// TwinCAT 3 PLC project Struckig
// Title: Struckig
// Company: Stefan Besler
// Author: Stefan Besler and contributers
// ProjectVersion: 0.6.0.0
// ProgramVersion: 3.1.4024.12
// CompilerDefines: ZEUGWERK_TWINCAT_3_1_4024_22
// project tree:
//   / Constants.TcGVL, ParameterList.TcGVL
//   Struckig/Block/ BlockInterval.TcDUT, Block.TcDUT
//   Struckig/BrakeProfile/ BrakeProfile.TcPOU
//   Struckig/ Integrate.TcPOU (not stored), Otg.TcPOU
//   Struckig/Math/ BubbleSortLreal.TcPOU, Ceil.TcPOU, LrealBits.TcPOU, LrealFromBits.TcPOU, Power.TcPOU, Power2.TcPOU, Cbrt.TcPOU, Roots.TcPOU
//   Struckig/Position/ PositionStep1.TcPOU, PositionStep2.TcPOU
//   Struckig/Profile/ ProfileDesc.TcPOU
//   Struckig/Profile/_DataTypes/ PositionExtremaDesc.TcDUT, ProfileDirection.TcDUT, ProfileJerkSigns.TcDUT, ProfileLimits.TcDUT
//   Struckig/Velocity/ VelocityStep1.TcPOU, VelocityStep2.TcPOU
//   Struckig/_DataTypes/ ControlInterfaceType.TcDUT, DiscretizationType.TcDUT, SynchronizationType.TcDUT, TrajectoryErrorCode.TcDUT, TrajectoryState.TcDUT

// ---- Struckig/Block/BlockInterval.TcDUT
/// Which times are possible for synchronization?
TYPE INTERNAL BlockInterval :
STRUCT
  IsUsed : BOOL;
  Left, Right : LREAL;
  Profile : ProfileDesc;
END_STRUCT
END_TYPE

// ---- Struckig/Block/Block.TcDUT
TYPE Block :
STRUCT
  p_min : ProfileDesc; // Save min Profile so that it doesn't need to be recalculated in Step2
  Tmin : LREAL; // [s]
  a, b : BlockInterval; // Max. 2 intervals can be blocked: called a and b with corresponding profiles, order does not matter  
END_STRUCT
END_TYPE

// ---- Struckig/Profile/_DataTypes/PositionExtremaDesc.TcDUT
TYPE PositionExtremaDesc :
STRUCT
  Minimum, Maximum : LREAL; // The extreme position
  Tmin, Tmax : LREAL;  // Time when the positions are reached
END_STRUCT
END_TYPE

// ---- Struckig/Profile/_DataTypes/ProfileDirection.TcDUT
{attribute 'qualified_only'}
{attribute 'strict'}
TYPE INTERNAL ProfileDirection :
(
  Up,
  Down
);
END_TYPE

// ---- Struckig/Profile/_DataTypes/ProfileJerkSigns.TcDUT
{attribute 'qualified_only'}
{attribute 'strict'}
TYPE ProfileJerkSigns :
(
	Uddu,
  Udud 
);
END_TYPE

// ---- Struckig/Profile/_DataTypes/ProfileLimits.TcDUT
{attribute 'qualified_only'}
{attribute 'strict'}
TYPE ProfileLimits :
(
	Acc0Acc1Vel,
  Vel, 
  Acc0,
  Acc1,
  Acc0Acc1,
  Acc0Vel,
  Acc1Vel,
  None
);
END_TYPE

// ---- Struckig/_DataTypes/ControlInterfaceType.TcDUT
{attribute 'qualified_only'}
{attribute 'strict'}
TYPE ControlInterfaceType :
(
  Position, // Position-control: Full control over the entire kinematic state (Default)
  Velocity // Velocity-control: Ignores the current position, target position, and velocity limits
);
END_TYPE

// ---- Struckig/_DataTypes/DiscretizationType.TcDUT
{attribute 'qualified_only'}
{attribute 'strict'}
TYPE DiscretizationType :
(
  Continuous, /// Every trajectory synchronization duration is allowed (Default)
  Discrete /// The trajectory synchronization duration must be a multiple of the control cycle
);
END_TYPE

// ---- Struckig/_DataTypes/SynchronizationType.TcDUT
{attribute 'qualified_only'}
{attribute 'strict'}
TYPE SynchronizationType :
(
  Undefined,
  Phase, // Phase synchronize the DoFs when possible, else fallback to "Time" strategy
  TimeSync, // Always synchronize the DoFs to reach the target at the same time (Default)
  TimeIfNecessarySync, // Synchronize only when necessary (e.g. for non-zero target velocity or acceleration)
  None // Calculate every DoF independently
);
END_TYPE

// ---- Struckig/_DataTypes/TrajectoryErrorCode.TcDUT
{attribute 'qualified_only'}
TYPE TrajectoryErrorCode :
(
	Undefined := 0,
  InvalidInput,
  SynchronizationFailed,
  CalculateStep1Failed
);
END_TYPE

// ---- Struckig/_DataTypes/TrajectoryState.TcDUT
{attribute 'qualified_only'}
{attribute 'strict'}
TYPE TrajectoryState :
(
  Undefined,
  Idle,
  Busy,
  Error
);
END_TYPE

// ---- Constants.TcGVL
{attribute 'qualified_only'}
VAR_GLOBAL INTERNAL CONSTANT
  BrakeEpsilon : LREAL := 2.2E-14;
  DoubleEpsilon : LREAL := 2.2204460492503131E-016; // smallest such that 1.0+Constants.DoubleEpsilon != 1.0
  DoubleEpsilonSqrt : LREAL := 1.483E-8;
  Epsilon : LREAL := 1E-8;
  Epsilon16 : LREAL := 16 * 1E-8;
  EpsilonColinear : LREAL := 1E-7;
  Infinity : LREAL := 1.7976931348623157E+308;  
  Tolerance : LREAL := 1E-14;
  Cos120 : LREAL := -0.50;
  Sin120 : LREAL := 0.866025403784438646764;  
  Pi : LREAL := 3.14159265358979323846;
  Minimum : LREAL := 1.17549435082E-38;  // used for validating input
END_VAR

// ---- ParameterList.TcGVL
{attribute 'qualified_only'}
VAR_GLOBAL CONSTANT
  MaxDoFs : INT := 7;
  MaxIterations : BYTE := 127; // Maximum iterations when [shrinking an interval](xref:Struckig.Roots#ShrinkInterval)
  NumericalRobust : BOOL := TRUE;
END_VAR

// ---- Struckig/Math/Roots.TcPOU
PROGRAM INTERNAL Roots
VAR
  a2, aover3, q, r2, q3, aa, t : LREAL;
  a, b, c, d, rr, theta, ux, uyi, inva, invaa, bb, bover3a, p, halfq, yy, inv2b, x, y, uuu, vvv, www, w, h : LREAL;
  discriminant : LREAL;
  e0, e1, q1, q2, p1, p2, dd, sqrtD  : LREAL;
  a3, b3, c3 : LREAL;
  x3 : ARRAY[0..2] OF LREAL;
  iZeroes : INT;  
  deriv : ARRAY[0 .. 10] OF LREAL;
  fl, fh, temp : LREAL;
  dxold, dx, f,df : LREAL;
  j : INT;
  xn : LREAL;
  iterations : BYTE;
END_VAR

METHOD PolyDeri
VAR_INPUT
  coeffs : POINTER TO LREAL;
  coeffsCount : BYTE;
  out : POINTER TO LREAL;
END_VAR
FOR j:=0 TO coeffsCount DO
  out[j] := (coeffsCount - j) * coeffs[j];
END_FOR
END_METHOD

METHOD PolyEval : LREAL;
VAR_INPUT
  polynom : POINTER TO LREAL;
  degree : INT;
  x : LREAL;
END_VAR
IF degree > 0 THEN
  IF (ABS(x) < Constants.DoubleEpsilon) THEN
      PolyEval := polynom[degree];
  ELSIF (x = 1.0) THEN
    FOR j:= degree TO 0 BY -1
    DO
      PolyEval := PolyEval + polynom[j];
    END_FOR
  ELSE
    xn := 1.0;
    FOR j:= degree TO 0 BY -1 
    DO
      PolyEval := PolyEval + polynom[j] * xn;
      xn := xn * x;
    END_FOR
  END_IF
END_IF
END_METHOD

METHOD PolyMonicDeri
VAR_INPUT
  monic_coeffs : POINTER TO LREAL;
  coeffsCount : BYTE;
  out : POINTER TO LREAL;  
END_VAR
VAR
  i : BYTE;
END_VAR
out[0] := 1.0;
FOR i:=1 TO coeffsCount-1 DO
  out[i] := (coeffsCount- i) * (monic_coeffs[i] / (coeffsCount));
END_FOR
END_METHOD

// Calculate a single zero of polynom p(x) inside [lbound, ubound]
// Requirements: p(lbound)*p(ubound) < 0, lbound < ubound
METHOD ShrinkInterval : LREAL
VAR_INPUT
  p : POINTER TO LREAL;
  degree : BYTE;  
  l, h : LREAL;
END_VAR
PolyDeri(p, degree, out:=ADR(deriv));
fl := PolyEval(p, degree, l);
fh := PolyEval(p, degree, h);
IF (fl = 0.0) THEN
  ShrinkInterval := l;
  RETURN;
END_IF

IF (fh = 0.0) THEN
  ShrinkInterval := h;
  RETURN;
END_IF

IF (fl > 0.0)
THEN
  // swap l and h
  temp := l;
  l := h;
  h := temp;
END_IF

ShrinkInterval := (l + h) / 2;
dxold := ABS(h - l);
dx := dxold;
f := PolyEval(p, degree, ShrinkInterval);
df := PolyEval(ADR(deriv), degree-1, ShrinkInterval);
FOR iterations:=0 TO ParameterList.MaxIterations DO
  IF ((((ShrinkInterval - h) * df - f) * ((ShrinkInterval - l) * df - f) > 0.0) OR_ELSE (ABS(2 * f) > ABS(dxold * df))) THEN
    dxold := dx;
    dx := (h - l) / 2;
    ShrinkInterval := l + dx;
    IF (l = ShrinkInterval) THEN
      RETURN;
    END_IF
  ELSE
    dxold := dx;
    dx := f / df;
    temp := ShrinkInterval;
    ShrinkInterval := ShrinkInterval - dx;
    IF (temp = ShrinkInterval) THEN
      RETURN;
    END_IF
  END_IF
  
  IF (ABS(dx) < Constants.Tolerance) THEN
    RETURN;
  END_IF
  
  f := PolyEval(p, degree, ShrinkInterval);
  df := PolyEval(ADR(deriv), degree-1, ShrinkInterval);
  IF (f < 0.0) THEN
    l := ShrinkInterval;
  ELSE
    h := ShrinkInterval;
  END_IF
END_FOR
END_METHOD

METHOD SolveCub
VAR_INPUT
  polynom : POINTER TO LREAL;
END_VAR
VAR_IN_OUT
  rootCount : INT;
  roots : ARRAY[0..6] OF LREAL;
END_VAR
rootCount := -1;
a := polynom[0];
b := polynom[1];
c := polynom[2];
d := polynom[3];

IF (ABS(d) < Constants.DoubleEpsilon)
THEN
  // First solution is x = 0
  roots[0] := 0.0;
  rootCount := 1;
  
  // Converting to a quadratic equation
  d := c;
  c := b;
  b := a;
  a := 0.0;
END_IF

IF (ABS(a) < Constants.DoubleEpsilon)
THEN
  IF (ABS(b) < Constants.DoubleEpsilon)
  THEN
    // Linear equation
    h := (-d / c);
    IF ABS(c) > Constants.DoubleEpsilon AND_THEN h >= 0
    THEN
      roots[rootCount+1] := h;
      rootCount := rootCount + 1;
    END_IF
  ELSE
    // Quadratic equation
    discriminant := c * c - 4 * b * d;
    IF (discriminant >= 0)
    THEN
      inv2b := 1.0 / (2 * b);
      y := SQRT(discriminant);
      
      h := ((-c + y) * inv2b);
      IF h >= 0
      THEN
        roots[rootCount+1] := h;
        rootCount := rootCount + 1;
			END_IF
      
      h := ((-c - y) * inv2b);
      IF h >= 0
      THEN      
        roots[rootCount+1] := ((-c - y) * inv2b);
        rootCount := rootCount + 1;
      END_IF
      
    END_IF
  END_IF

ELSE
  
  // Cubic equation
  inva := 1.0 / a;
  invaa := inva * inva;
  bb := b * b;
  bover3a := b * inva / 3;
  p := (a * c - bb / 3) * invaa;
  halfq := (2 * bb * b - 9 * a * b * c + 27 * a * a * d) * (0.5 / 27) * invaa * inva;
  yy := p * p * p / 27 + halfq * halfq;  
    
  IF (yy > Constants.DoubleEpsilon) THEN
    // Sqrt is positive: one real solution}
    y := SQRT(yy);
    uuu := -halfq + y;
    vvv := -halfq - y;
    www := SEL(ABS(uuu) > ABS(vvv), vvv, uuu);
    w := cbrt(www);
    
    h := (w - p / (3 * w) - bover3a);
    IF h >= 0
    THEN
      roots[rootCount+1] := h;
      rootCount := rootCount + 1;    
		END_IF

  ELSIF (yy < -Constants.DoubleEpsilon) THEN
    // Sqrt is negative: three real solutions
    x := -halfq;
    y := SQRT(-yy);

    // Convert to polar form}
    IF ABS(x) > Constants.DoubleEpsilon THEN
      theta := SEL((x > 0.0), (ATAN(y / x) + Constants.Pi), ATAN(y / x));
      rr := SQRT(x * x - yy);
    ELSE
      // Vertical line}
      theta := Constants.Pi / 2;
      rr := y;
    END_IF
    
    // Calculate cube root
    theta := theta / 3;
    rr := 2 * cbrt(rr);
    // Convert to complex coordinate
    ux := COS(theta) * rr;
    uyi := SIN(theta) * rr;
    // First solution
    h := (ux - bover3a);
    IF h >= 0
    THEN
      roots[rootCount+1] := h;
      rootCount := rootCount + 1;
		END_IF
    
    // Second solution, rotate +120 degrees
    h := ux * Constants.Cos120 - uyi * Constants.Sin120 - bover3a;
    IF h >= 0
    THEN
      roots[rootCount+1] := h;
      rootCount := rootCount + 1;
		END_IF
    
    // Third solution, rotate -120 degrees
    h := ux * Constants.Cos120 + uyi * Constants.Sin120 - bover3a;
    IF h >= 0
    THEN
      roots[rootCount+1] := h;
      rootCount := rootCount + 1;
		END_IF
  ELSE
    // Sqrt is zero: two real solutions
    www := -halfq;
    w := 2 * cbrt(www);
    // First solution
    h := (w - bover3a);
    IF h >= 0
    THEN
      roots[rootCount+1] := h;
      rootCount := rootCount + 1;
		END_IF
    
    // Second solution, rotate +120 degrees
    h := (w * Constants.Cos120 - bover3a);
    IF h >= 0
    THEN
      roots[rootCount+1] := h;
      rootCount := rootCount + 1;
		END_IF
  END_IF
END_IF
END_METHOD

/// Calculate all roots of the monic quartic equation: x^4 + a*x^3 + b*x^2 + c*x + d = 0
METHOD SolveQuartMonic
VAR_INPUT
  polynom : POINTER TO LREAL;  
  degree : LREAL;
END_VAR
VAR_IN_OUT
  rootCount : INT;
  roots : ARRAY[0..6] OF LREAL;
END_VAR
rootCount := -1;

a := polynom[0];
b := polynom[1];
c := polynom[2];
d := polynom[3];
e0 := cbrt(c * c);
IF (ABS(a) < Constants.DoubleEpsilon AND_THEN ABS(b) < Constants.DoubleEpsilonSqrt AND_THEN ABS(c) < Constants.DoubleEpsilonSqrt AND_THEN ABS(d) < Constants.DoubleEpsilon) AND_THEN
   ABS(e0) > Constants.DoubleEpsilon
THEN
  e1 := (b * b + 12 * d)/(9 * e0);
  q1 := -(4 * b) / 3 - e0 - e1;
  p1 := SQRT(-q1 - 2 * b);
  q2 := 2 * c / p1;
  
  dd := q1 - q2;
  IF (dd > 0.0)
  THEN  
    sqrtD := SQRT(dd);
    
    h := ((p1 + sqrtD) / 2);
    IF h >= 0
    THEN
      roots[0] := h;
      rootCount := 0;
		END_IF
    
    h := ((p1 - sqrtD) / 2);
    IF h >= 0
    THEN
      roots[rootCount+1] := h;
      rootCount := rootCount + 1;
		END_IF
  END_IF
  
  dd := q1 + q2;
  IF (dd > 0.0)
  THEN  
    sqrtD := SQRT(dd);
    
    h := ((-p1 + sqrtD) / 2);
    IF h >= 0
    THEN
      roots[rootCount+1] := h;
      rootCount := rootCount + 1;
		END_IF
    
    h := ((-p1 - sqrtD) / 2);
    IF h >= 0
    THEN
      roots[rootCount+1] := h;
      rootCount := rootCount + 1;
		END_IF
  END_IF
  RETURN;
END_IF

IF (ABS(c) < Constants.DoubleEpsilon AND_THEN ABS(d) < Constants.DoubleEpsilon)
THEN
  roots[0] := 0.0;
  rootCount := rootCount+1;
  
  dd := a * a - 4 * b;
  IF (ABS(dd) < Constants.DoubleEpsilon)
  THEN
    h := (-a / 2);
    IF h >= 0
    THEN
      roots[rootCount+1] := h;
      rootCount := rootCount + 1;
		END_IF
  ELSIF (dd > 0)
  THEN
    sqrtD := SQRT(dd);
    h := ((-a - sqrtD) / 2);
    IF h >= 0
    THEN
      roots[rootCount+1] := h;
      rootCount := rootCount + 1;
		END_IF
    
    h := ((-a + sqrtD) / 2);
    IF h >= 0
    THEN
      roots[rootCount+1] := h;
      rootCount := rootCount + 1;
		END_IF  
  END_IF
  RETURN;
END_IF

a3 := -b;
b3 := a * c - 4 * d;
c3 := -a * a * d - c * c + 4 * b * d;

// Solve the resolvent: y^3 - b*y^2 + (ac - 4*d)*y - a^2*d - c^2 + 4*b*d = 0
iZeroes := SolveResolvent(ADR(x3), a3, b3, c3);

y := x3[0];
// Choosing Y with maximal absolute value.
IF (iZeroes <> 1) THEN
  IF ABS(x3[1]) > ABS(y) THEN
    y := x3[1];
  END_IF
  
  IF ABS(x3[2]) > ABS(y) THEN
    y := x3[2];
  END_IF
END_IF

// h1 + h2 = y AND_THEN h1*h2 = d  <=>  h^2 - y*h + d = 0    (h === q)
dd := y * y - 4 * d;
IF (ABS(dd) < Constants.DoubleEpsilon) THEN
  q1 := q2 := y / 2;
  // g1 + g2 = a AND_THEN g1 + g2 = b - y   <=>   g^2 - a*g + b - y = 0    (p === g)}
  dd := a * a - 4 * (b - y);
  IF (ABS(dd) < Constants.DoubleEpsilon) THEN
    p1 := p2 := a / 2;
  ELSE
    sqrtD := SQRT(dd);
    p1 := (a + sqrtD) / 2;
    p2 := (a - sqrtD) / 2;
  END_IF
ELSE
  sqrtD := SQRT(dd);
  q1 := (y + sqrtD) / 2;
  q2 := (y - sqrtD) / 2;
  // g1 + g2 = a AND_THEN g1*h2 + g2*h1 = c   ( AND_THEN g === p )  Krammer
  p1 := (a * q1 - c) / (q1 - q2);
  p2 := (c - a * q2) / (q1 - q2);
END_IF

// Solve the quadratic equation: x^2 + p1*x + q1 = 0
dd := p1 * p1 - 4 * q1;
IF (ABS(dd) < Constants.Epsilon16) THEN
  
  h:= (-p1 / 2);
  IF h >= 0
  THEN
    roots[rootCount+1] := h;
    rootCount := rootCount + 1;
  END_IF
  
ELSIF (dd > 0.0)  THEN
  sqrtD := SQRT(dd);
  h := ((-p1 + sqrtD) / 2);
  IF h >= 0
  THEN
    roots[rootCount+1] := h;
    rootCount := rootCount + 1;
  END_IF
    
  h := ((-p1 - sqrtD) / 2);
  IF h >= 0
  THEN
    roots[rootCount+1] := h;
    rootCount := rootCount + 1;
  END_IF
END_IF

// Solve the quadratic equation: x^2 + p2*x + q2 = 0
dd := p2 * p2 - 4 * q2;
IF (ABS(dd) < Constants.Epsilon16) THEN
  h := (-p2 * 0.5);
  IF h >= 0
  THEN
    roots[rootCount+1] := h;
    rootCount := rootCount + 1;
  END_IF  
ELSIF (dd > 0.0) THEN
  sqrtD := SQRT(dd);
  h := ((-p2 + sqrtD) / 2); 
  IF h >= 0
  THEN
    roots[rootCount+1] := h;
    rootCount := rootCount + 1;
  END_IF
  
  h := ((-p2 - sqrtD) / 2);
  IF h >= 0
  THEN
    roots[rootCount+1] := h;
    rootCount := rootCount + 1;
  END_IF
END_IF
END_METHOD

/// Solve resolvent eqaution of corresponding Quartic equation
/// The input x must be of length 3
/// Number of zeros are returned
METHOD SolveResolvent : INT
VAR_INPUT
  x : POINTER TO LREAL;
  a,b,c : LREAL;
END_VAR
aover3 := a / 3;
a2 := a * a;
q := (a2 - 3 * b) / 9;
rr := a * (2 * a2 - 9 * b) / 54 + c / 2;
r2 := rr * rr;
q3 := q * q * q;

IF (r2 < q3) THEN
  t := rr / SQRT(q3);
  IF (t < -1.0) THEN
      t := -1.0;
  END_IF
  
  IF (t > 1.0) THEN
      t := 1.0;
  END_IF
  
  q := -2 * SQRT(q);
  theta := ACOS(t) / 3;
  ux := COS(theta) * q;
  uyi := SIN(theta) * q;
  x[0] := ux - aover3;
  x[1] := ux * Constants.Cos120 - uyi * Constants.Sin120 - aover3;
  x[2] := ux * Constants.Cos120 + uyi * Constants.Sin120 - aover3;
  SolveResolvent := 3;
  RETURN;

ELSE
  aa := -cbrt(ABS(rr) + SQRT(r2 - q3));
  IF (rr < 0.0) THEN
    aa := -aa;
  END_IF
  bb := SEL(0.0 = aa, q / aa, 0.0);
  
  x[0] := (aa + bb) - aover3;
  x[1] := -(aa + bb) / 2 - aover3;
  x[2] := SQRT(3) * (aa - bb) / 2;
  IF (ABS(x[2]) < Constants.DoubleEpsilon) THEN
    x[2] := x[1];
    SolveResolvent := 2;
    RETURN;
  END_IF
  
  SolveResolvent := 1;
END_IF
END_METHOD

END_PROGRAM

// ---- Struckig/Math/Cbrt.TcPOU
/// The TwinCAT code is a modified version of the original C code from
/// http://www.netlib.org/fdlibm/s_cbrt.c and came with this notice.
///
/// ```
/// Copyright (C) 1993 by Sun Microsystems, Inc. All rights reserved.
///
/// Developed at SunSoft, a Sun Microsystems, Inc. business.
/// Permission to use, copy, modify, and distribute this
/// software is freely granted, provided that this notice
/// is preserved.
/// ```
///
///
/// Small modifications were made, while the original code said
/// ```
/// chop to 20 bits, make larger than cbrt(x)
/// t := LrealFromBits((LrealBits(t) AND SHL(H, 28)) + SHL(J, 30));
/// ```
/// Modern compilers seem to round t away from 0 to 23 bits.
/// see https://github.com/stdlib-js/math-base-special-cbrt/blob/main/src/cbrt.c
FUNCTION Cbrt : LREAL
VAR_INPUT
  x : LREAL;
END_VAR
VAR CONSTANT
  B1 : ULINT := 715094163;                  // (682-0.03306235651)*2**20
  B2 : ULINT := 696219795;                  // (664-0.03306235651)*2**20
  C : LREAL := 5.42857142857142815906E-01;  // 19/35     = 0x3FE15F15F15F15F1
  D : LREAL := -7.05306122448979611050E-01; // -864/1225 = 0xBFE691DE2532C834
  E : LREAL := 1.41428571428571436819E+00;  // 99/70     = 0x3FF6A0EA0EA0EA0F
  F : LREAL := 1.60714285714285720630E+00;  // 45/28     = 0x3FF9B6DB6DB6DB6E
  G : LREAL := 3.57142857142857150787E-01;  // 5/14      = 0x3FD6DB6DB6DB6DB7
  J : ULINT := 1;
  Mask : ULINT := ULINT#16#FFFFFFFFC0000000;
  AMask : ULINT := ULINT#16#80000000;
  SmallestNormal : LREAL := 2.22507385850720138309E-308; // 2**-1022  = 0x0010000000000000  
END_VAR
VAR
  sign : BOOL;
  t, r1, s1, w : LREAL;
END_VAR

// test x=0 and x=NaN
IF x = 0 OR_ELSE x <> x
THEN
  Cbrt := x;
  RETURN;
END_IF

sign := FALSE;
IF x < 0
THEN
  x := -x;
  sign := TRUE;  
END_IF

// rough cbrt to 5 bits
t := LrealFromBits(LrealBits(x)/3 + SHL(B1, 32));
IF x < SmallestNormal
THEN
  // subnormal number
  t := LrealFromBits(SHL(J, 54)); // set t= 2**54
  t := t * x;
  t := LrealFromBits(LrealBits(t)/3 + SHL(B2, 32));
END_IF

// new cbrt to 23 bits
r1 := t * t / x;
s1 := C + r1*t;
t := t * (G + F/(s1+E+D/s1));

// see https://github.com/stdlib-js/math-base-special-cbrt/blob/main/src/cbrt.c
t := LrealFromBits((LrealBits(t) + AMask) AND Mask);

// one step newton iteration to 53 bits with error less than 0.667ulps
s1 := t * t; // t*t is exact
r1 := x / s1;
w := t + t;
r1 := (r1 - t) / (w + r1); // r-s is exact
t := t + t*r1;

// restore the sign bit
IF sign
THEN
  t := -t;
END_IF

Cbrt := t;
    
// this one is a bit more prone to numerical errors
// Cbrt := SEL(x < 0, 1.0, -1.0) * EXPT(ABS(x), 1.0 / 3.0);

END_FUNCTION

// ---- Struckig/Math/LrealFromBits.TcPOU
{attribute 'hide'}
FUNCTION LrealFromBits : LREAL
VAR_INPUT
  b : ULINT;
END_VAR
VAR
  x : POINTER TO LREAL := ADR(b);
END_VAR

LrealFromBits := x^;

END_FUNCTION

// ---- Struckig/Math/LrealBits.TcPOU
{attribute 'hide'}
FUNCTION LrealBits : ULINT
VAR_INPUT
  x : LREAL;
END_VAR
VAR
  b : POINTER TO ULINT := ADR(x);
END_VAR

LrealBits := b^;

END_FUNCTION

// ---- Struckig/BrakeProfile/BrakeProfile.TcPOU
/// Calculates (pre- or post-) profile to get current or final state below the limits
FUNCTION_BLOCK BrakeProfile
VAR_INPUT
  Duration : LREAL; //! Overall duration
  t, j, a, v, p : ARRAY[0..1] OF LREAL; //! Profile information for a two-step profile  
  IsUsed : BOOL;
END_VAR
VAR
  t_to_a_min, t_to_a_max, t_min_to_v_max, t_to_a_zero, t_to_v_min, t_to_v_max : LREAL;
  t_to_v_max_with_constant, t_to_v_min_with_constant, v_at_a0, v_at_a_max, v_at_a_min : LREAL;
END_VAR

METHOD AccelerationBrake
VAR_INPUT
  v0, a0 : LREAL;
  vMax, vMin : LREAL;
  aMax, aMin : LREAL;
  jMax : LREAL;
END_VAR
VAR_IN_OUT
  t_brake : ARRAY[0..1] OF LREAL;
  j_brake : ARRAY[0..1] OF LREAL;    
END_VAR
j_brake[0] := -jMax;

t_to_a_max := (a0 - aMax) / jMax;
t_to_a_zero := a0 / jMax;

v_at_a_max := VelocityAtTime(v0, a0, -jMax, t_to_a_max);
v_at_a0 := VelocityAtTime(v0, a0, -jMax, t_to_a_zero);

IF (v_at_a0 > vMax AND_THEN jMax > 0) OR_ELSE (v_at_a0 < vMax AND_THEN jMax < 0)
THEN
  VelocityBrake(v0, a0, vMax, vMin, aMax, aMin, jMax, t_brake, j_brake);

ELSIF (v_at_a_max < vMin AND_THEN jMax > 0) OR_ELSE (v_at_a_max > vMin AND_THEN jMax < 0)
THEN
  t_to_v_min := -(v_at_a_max - vMin)/aMax;
  t_to_v_max := -aMax/(2*jMax) - (v_at_a_max + vMax)/aMax;
  t_brake[0] := t_to_a_max + Constants.BrakeEpsilon;
  t_brake[1] := MAX(MIN(t_to_v_min, v_at_a_max - Constants.BrakeEpsilon), 0.0);
ELSE
  t_brake[0] := t_to_a_max + Constants.BrakeEpsilon;
END_IF
END_METHOD

METHOD PositionBrakeTrajectory
VAR_INPUT
  v0, a0 : LREAL;
  vMax, vMin : LREAL;
  aMax, aMin : LREAL;
  jMax : LREAL;
END_VAR
VAR_IN_OUT
  t_brake : ARRAY[0..1] OF LREAL;
  j_brake : ARRAY[0..1] OF LREAL;    
END_VAR
t_brake[0] := 0.0;
t_brake[1] := 0.0;
j_brake[0] := 0.0;
j_brake[1] := 0.0;

IF a0 > aMax
THEN
  AccelerationBrake(v0, a0, vMax, vMin, aMax, aMin, jMax, t_brake, j_brake);
ELSIF a0 < aMin
THEN
  AccelerationBrake(v0, a0, vMin, vMax, aMin, aMax, -jMax, t_brake, j_brake);
ELSIF ((v0 > vMax AND_THEN VelocityAtZeroAcceleration(v0, a0, -jMax) > vMin) OR_ELSE (a0 > 0 AND_THEN VelocityAtZeroAcceleration(v0, a0, jMax) > vMax))
THEN
  VelocityBrake(v0, a0, vMax, vMin, aMax, aMin, jMax, t_brake, j_brake);
ELSIF ((v0 < vMin AND_THEN VelocityAtZeroAcceleration(v0, a0, jMax) < vMax) OR_ELSE (a0 < 0 AND_THEN VelocityAtZeroAcceleration(v0, a0, -jMax) < vMin))
THEN
  VelocityBrake(v0, a0, vMin, vMax, aMin, aMax, -jMax, t_brake, j_brake);      
END_IF
END_METHOD

METHOD VelocityAtTime : LREAL
VAR_INPUT
  v0, a0 : LREAL;
  j : LREAL;
  t : LREAL;
END_VAR
VelocityAtTime := v0 + t * (a0 + j * t * 0.5);
END_METHOD

METHOD VelocityAtZeroAcceleration : LREAL
VAR_INPUT
  v0, a0 : LREAL;
  j : LREAL;
END_VAR
VelocityAtZeroAcceleration := v0 + (a0 * a0) / (2 * j);
END_METHOD

METHOD VelocityBrake
VAR_INPUT
  v0, a0 : LREAL;
  vMax, vMin : LREAL;
  aMax, aMin : LREAL;
  jMax : LREAL;
END_VAR
VAR_IN_OUT
  t_brake : ARRAY[0..1] OF LREAL;
  j_brake : ARRAY[0..1] OF LREAL;    
END_VAR
j_brake[0] := -jMax;
t_to_a_min := (a0 - aMin)/jMax;
t_to_v_max := a0*a0 + 2 * jMax * (v0 - vMax);
t_to_v_min := a0*a0 / 2 + jMax * (v0 - vMin);

IF t_to_v_max < 0 OR_ELSE t_to_v_min < 0
THEN
  RETURN;
END_IF

t_to_v_max := a0/jMax + SQRT(t_to_v_max) / ABS(jMax);
t_to_v_min := a0/jMax + SQRT(t_to_v_min) / ABS(jMax);
t_min_to_v_max := MIN(t_to_v_max, t_to_v_min);

IF (t_to_a_min < t_min_to_v_max)
THEN
  v_at_a_min := VelocityAtTime(v0, a0, -jMax, t_to_a_min);
  t_to_v_max_with_constant := -(v_at_a_min - vMax)/aMin;
  t_to_v_min_with_constant := -0.5*aMin/jMax - (v_at_a_min - vMin)/aMin;
  t_brake[0] := t_to_a_min - Constants.BrakeEpsilon;
  t_brake[1] := MAX(MIN(t_to_v_max_with_constant, t_to_v_min_with_constant), 0.0);
ELSE
  t_brake[0] := t_min_to_v_max - Constants.BrakeEpsilon;
END_IF
END_METHOD

METHOD VelocityBrakeTrajectory
VAR_INPUT
  v0, a0 : LREAL;
  aMax, aMin : LREAL;
  jMax : LREAL;
END_VAR
VAR_IN_OUT
  t_brake : ARRAY[0..1] OF LREAL;
  j_brake : ARRAY[0..1] OF LREAL;    
END_VAR
t_brake[0] := 0.0;
t_brake[1] := 0.0;
j_brake[0] := 0.0;
j_brake[1] := 0.0;

IF (a0 > aMax)
THEN
  j_brake[0] := -jMax;
  t_brake[0] := (a0 - aMax)/jMax + Constants.BrakeEpsilon;
ELSIF (a0 < aMin)
THEN
  j_brake[0] := jMax;
  t_brake[0] := -(a0 - aMin)/jMax + Constants.BrakeEpsilon;
END_IF
END_METHOD

END_FUNCTION_BLOCK

// ---- Struckig/Math/BubbleSortLreal.TcPOU
FUNCTION BubbleSortLreal : BOOL
VAR_INPUT
  data : POINTER TO LREAL; // input unsorted array
  size : INT; // elements in the data array
  indicesSorted : POINTER TO INT; // actual output, sorted indices
END_VAR
VAR
  i, j, h : INT;
END_VAR

FOR i:=0 TO size
DO
  indicesSorted[i] := i;
END_FOR

// Bubblesort possible_t_syncs from best to worst
FOR i:=0 TO size-1
DO
  FOR j:=0 TO size-1-i
  DO  
    IF data[indicesSorted[j]] > data[indicesSorted[j+1]]
    THEN
      h := indicesSorted[j];
      indicesSorted[j] := indicesSorted[j+1];
      indicesSorted[j+1] := h;     
		END_IF
  END_FOR
END_FOR

END_FUNCTION

// ---- Struckig/Math/Ceil.TcPOU
FUNCTION Ceil : LREAL
VAR_INPUT
  val : LREAL;
END_VAR
VAR CONSTANT
  InfinityBits : ULINT := ULINT#16#7FF0000000000000;
END_VAR
VAR
  InfinityPtr : POINTER TO LREAL := ADR(InfinityBits);
END_VAR

IF val <> val OR_ELSE val = InfinityPtr^ OR_ELSE val = -InfinityPtr^ // nan or inf
THEN
  RETURN;
END_IF

Ceil := DINT_TO_LREAL(LREAL_TO_DINT(val));
IF Ceil < val THEN
	Ceil := Ceil + 1;
END_IF;

END_FUNCTION

// ---- Struckig/Math/Power.TcPOU
FUNCTION INTERNAL Power : LREAL
VAR_INPUT
  v : LREAL;
  e : LREAL;
END_VAR

Power := SEL(v < 0, 1.0, -1.0) * EXPT(ABS(v), e);

END_FUNCTION

// ---- Struckig/Math/Power2.TcPOU
FUNCTION INTERNAL Power2 : LREAL
VAR_INPUT
  v : LREAL;
END_VAR

Power2 := v*v;

END_FUNCTION

// ---- Struckig/Position/PositionStep1.TcPOU
FUNCTION_BLOCK INTERNAL PositionStep1
VAR
  p0, v0, a0 : LREAL;
  pf, vf, af : LREAL;
  _vMax, _vMin, _aMax, _aMin, _jMax : LREAL;

  // Pre-calculated expressions
  pd : LREAL;
  v0_v0, vf_vf : LREAL;
  a0_a0, a0_p3, a0_p4 : LREAL;
  af_af, af_p3, af_p4 : LREAL;
  jMax_jMax : LREAL;
  
  // runtime  calculated expressions
  polynom : ARRAY[0..4] OF LREAL;
  orig : LREAL;
  deriv : LREAL;
  t : LREAL;
  i : INT;
  h0, h1, h2, h2_h2, h3 : LREAL;
  t_min, t_max : LREAL;
  t_acc1, t_acc0 : LREAL;
  validProfiles : ARRAY[0..5] OF ProfileDesc; // Max 5 valid profiles + 1 spare for numerical issues
  validProfileCounter : INT := -1;
  
  rootCount : INT;
  root : ARRAY[0..6] OF LREAL;
  left_duration, right_duration : LREAL;   
END_VAR

METHOD AddInterval
VAR_INPUT
  interval : REFERENCE TO BlockInterval;
  Left : REFERENCE TO ProfileDesc;
  Right : REFERENCE TO ProfileDesc;
END_VAR
left_duration := Left.t_sum[6] + Left.Brake.Duration;
right_duration := Right.t_sum[6] + Right.Brake.Duration;
IF (left_duration < right_duration)
THEN
  interval.Left := left_duration;
  interval.Right := right_duration;
  interval.Profile := Right;
  interval.IsUsed := TRUE;
ELSE
  interval.Left := right_duration;
  interval.Right := left_duration;
  interval.Profile := Left;
  interval.IsUsed := TRUE;  
END_IF
END_METHOD

METHOD AddProfile
VAR_IN_OUT CONSTANT
  Profile : ProfileDesc;
  jMax : LREAL;
END_VAR
validProfileCounter := validProfileCounter + 1;
validProfiles[validProfileCounter] := Profile;
validProfiles[validProfileCounter].Direction := SEL(jMax > 0, ProfileDirection.Down, ProfileDirection.Up);
END_METHOD

METHOD CalculateBlock : BOOL
VAR_INPUT
  block : REFERENCE TO Block;
END_VAR
VAR
  i, j : INT;
  Tmin : LREAL;
  idx_min : INT;
  idx_else_1, idx_else_2, idx_else_3, idx_else_4 : INT;
END_VAR
IF validProfileCounter = 0
THEN
  block.Pmin := validProfiles[0];
  block.Tmin := block.Pmin.t_sum[6] + block.Pmin.Brake.Duration;  
  CalculateBlock := TRUE;

ELSIF validProfileCounter = 1 
THEN

  IF ABS(validProfiles[0].t_sum[6] - validProfiles[1].t_sum[6]) < 8*Constants.Epsilon
  THEN
    block.Pmin := validProfiles[0];
    block.Tmin := block.Pmin.t_sum[6] + block.Pmin.Brake.Duration;  
    CalculateBlock := TRUE;
    RETURN;
	END_IF
  
  IF ParameterList.NumericalRobust
  THEN
    idx_min := SEL(validProfiles[0].t_sum[6] < validProfiles[1].t_sum[6], 1, 0);
    idx_else_1 := (idx_min + 1) MOD 2;

    block.Pmin := validProfiles[idx_min];
    block.Tmin := block.Pmin.t_sum[6] + block.Pmin.Brake.Duration;
    
    AddInterval(block.A, validProfiles[idx_min], validProfiles[idx_else_1]);
    CalculateBlock := TRUE;
    RETURN; 
	END_IF

// Only happens due to numerical issues
ELSIF (validProfileCounter = 3) 
THEN
  // Find "identical" profiles
  IF (ABS(validProfiles[0].t_sum[6] - validProfiles[1].t_sum[6]) < 32*Constants.Epsilon AND_THEN validProfiles[0].Direction <> validProfiles[1].Direction)
  THEN
    RemoveProfile(1);
  ELSIF (ABS(validProfiles[2].t_sum[6] - validProfiles[3].t_sum[6]) < 256*Constants.Epsilon  AND_THEN validProfiles[2].Direction <> validProfiles[3].Direction)
  THEN
    RemoveProfile(3);
  ELSIF (ABS(validProfiles[0].t_sum[6] - validProfiles[3].t_sum[6]) < 256*Constants.Epsilon AND_THEN validProfiles[0].Direction <> validProfiles[3].Direction)
  THEN
    RemoveProfile(3);
  ELSE
    RETURN;
  END_IF

ELSIF ((validProfileCounter+1) MOD 2 = 0)
THEN
  RETURN;
END_IF

// Find index of fastest Profile
Tmin := Constants.Infinity;
FOR i:=0 TO validProfileCounter
DO
  FOR j:=0 TO validProfileCounter
  DO
    IF validProfiles[i].t_sum[6] + validProfiles[i].brake.Duration < validProfiles[j].t_sum[6] + validProfiles[j].brake.Duration AND_THEN
       validProfiles[i].t_sum[6] + validProfiles[i].brake.Duration < Tmin
    THEN
      Tmin := validProfiles[i].t_sum[6] + validProfiles[i].brake.Duration;
      idx_min := i;
		END_IF
  END_FOR
END_FOR

block.A.IsUsed := FALSE;
block.B.IsUsed := FALSE;
block.Pmin := validProfiles[idx_min];
block.Tmin := block.Pmin.t_sum[6] + block.Pmin.Brake.Duration;  

IF (validProfileCounter = 2)
THEN
  idx_else_1 := (idx_min + 1) MOD 3;
  idx_else_2 := (idx_min + 2) MOD 3;
  
  AddInterval(block.A, validProfiles[idx_else_1], validProfiles[idx_else_2]);
  CalculateBlock := TRUE;
  RETURN;

 ELSIF (validProfileCounter = 4)
 THEN
  idx_else_1 := (idx_min + 1) MOD 5;
  idx_else_2 := (idx_min + 2) MOD 5;
  idx_else_3 := (idx_min + 3) MOD 5;
  idx_else_4 := (idx_min + 4) MOD 5;
  
  IF (validProfiles[idx_else_1].Direction = validProfiles[idx_else_2].Direction)
  THEN
    AddInterval(block.A, validProfiles[idx_else_1], validProfiles[idx_else_2]);
    AddInterval(block.B, validProfiles[idx_else_3], validProfiles[idx_else_4]);
  ELSE 
    AddInterval(block.A, validProfiles[idx_else_1], validProfiles[idx_else_4]);
    AddInterval(block.B, validProfiles[idx_else_2], validProfiles[idx_else_3]);
  END_IF
  
  CalculateBlock := TRUE;
END_IF
END_METHOD

METHOD Get : BOOL
VAR_INPUT
  Profilefile : REFERENCE TO ProfileDesc;
  block : REFERENCE TO Block; 
END_VAR
VAR_INST
  vMax, vMin, aMax, aMin, jMax : LREAL;  
END_VAR
Profilefile.SetBoundaryPosition(p0, v0, a0, pf, vf, af);
validProfileCounter := -1;

IF (ABS(vf) < Constants.DoubleEpsilon AND_THEN ABS(af) < Constants.DoubleEpsilon) THEN
  vMax := SEL(pd >= 0, _vMin, _vMax);
  vMin := SEL(pd >= 0, _vMax, _vMin);
  aMax := SEL(pd >= 0, _aMin, _aMax);
  aMin := SEL(pd >= 0, _aMax, _aMin);
  jMax :=SEL (pd >= 0,-_jMax, _jMax);

  IF ABS(v0) < Constants.DoubleEpsilon AND_THEN ABS(a0) < Constants.DoubleEpsilon AND_THEN ABS(pd) < Constants.DoubleEpsilon
  THEN
    time_none(Profilefile, vMax, vMin, aMax, aMin, jMax);
  ELSE
    // There is no blocked interval when vf==0 && af==0, so return after first found profile
    time_all_vel(Profilefile, vMax, vMin, aMax, aMin, jMax);
    IF (validProfileCounter > 0) THEN
      Get := CalculateBlock(block);
      RETURN;
    END_IF
    time_none(Profilefile, vMax, vMin, aMax, aMin, jMax);
    IF (validProfileCounter > 0) THEN
      Get := CalculateBlock(block);
      RETURN;
    END_IF
    time_acc0(Profilefile, vMax, vMin, aMax, aMin, jMax);
    IF (validProfileCounter > 0) THEN
      Get := CalculateBlock(block);
      RETURN;
    END_IF
    time_acc1(Profilefile, vMax, vMin, aMax, aMin, jMax);
    IF (validProfileCounter > 0) THEN
      Get := CalculateBlock(block);
      RETURN;
    END_IF
    time_acc0_acc1(Profilefile, vMax, vMin, aMax, aMin, jMax);
    IF (validProfileCounter > 0) THEN
      Get := CalculateBlock(block);
      RETURN;
    END_IF
    time_all_vel(Profilefile, vMax, vMin, aMax, aMin, jMax);
    IF (validProfileCounter > 0) THEN
      Get := CalculateBlock(block);
      RETURN;
    END_IF
    time_none(Profilefile, vMin, vMax, aMin, aMax, -jMax);
    IF (validProfileCounter > 0) THEN
      Get := CalculateBlock(block);
      RETURN;
    END_IF
    time_acc0(Profilefile, vMin, vMax, aMin, aMax, -jMax);
    IF (validProfileCounter > 0) THEN
      Get := CalculateBlock(block);
      RETURN;
    END_IF
    time_acc1(Profilefile, vMin, vMax, aMin, aMax, -jMax);
    IF (validProfileCounter > 0) THEN
      Get := CalculateBlock(block);
      RETURN;
    END_IF
    time_acc0_acc1(Profilefile, vMin, vMax, aMin, aMax, -jMax);          
  END_IF
ELSE 
  time_all_vel(Profilefile, _vMax, _vMin, _aMax, _aMin, _jMax);
  time_all_vel(Profilefile, _vMin, _vMax, _aMin, _aMax, -_jMax);
  time_none(Profilefile, _vMax, _vMin, _aMax, _aMin, _jMax);
  time_acc0(Profilefile, _vMax, _vMin, _aMax, _aMin, _jMax);
  time_acc1(Profilefile, _vMax, _vMin, _aMax, _aMin, _jMax);
  time_acc0_acc1(Profilefile, _vMax, _vMin, _aMax, _aMin, _jMax);
  time_none(Profilefile, _vMin, _vMax, _aMin, _aMax, -_jMax);
  time_acc0(Profilefile, _vMin, _vMax, _aMin, _aMax, -_jMax);
  time_acc1(Profilefile, _vMin, _vMax, _aMin, _aMax, -_jMax);
  time_acc0_acc1(Profilefile, _vMin, _vMax, _aMin, _aMax, -_jMax);  
END_IF

IF (validProfileCounter = -1)
THEN
  time_none_two_step(Profilefile, _vMax, _vMin, _aMax, _aMin, _jMax);
  IF validProfileCounter >= 0
  THEN
    Get := CalculateBlock(block);
    RETURN;
	END_IF
  
  time_none_two_step(Profilefile, _vMin, _vMax, _aMin, _aMax, -_jMax);
  IF validProfileCounter >= 0
  THEN
    Get := CalculateBlock(block);
    RETURN;
	END_IF
  

  time_acc0_two_step(Profilefile, _vMax, _vMin, _aMax, _aMin, _jMax);
  IF validProfileCounter >= 0
  THEN
    Get := CalculateBlock(block);
    RETURN;
	END_IF
  
  time_acc0_two_step(Profilefile, _vMin, _vMax, _aMin, _aMax, -_jMax);
  IF validProfileCounter >= 0
  THEN
    Get := CalculateBlock(block);
    RETURN;
	END_IF
  
  time_vel_two_step(Profilefile, _vMax, _vMin, _aMax, _aMin, _jMax);
  IF validProfileCounter >= 0
  THEN
    Get := CalculateBlock(block);
    RETURN;
	END_IF
  
  time_vel_two_step(Profilefile, _vMin, _vMax, _aMin, _aMax, -_jMax);
  IF validProfileCounter >= 0
  THEN
    Get := CalculateBlock(block);
    RETURN;
	END_IF
  
  time_acc1_vel_two_step(Profilefile, _vMax, _vMin, _aMax, _aMin, _jMax);
  IF validProfileCounter >= 0
  THEN
    Get := CalculateBlock(block);
    RETURN;
	END_IF
  
  time_acc1_vel_two_step(Profilefile, _vMin, _vMax, _aMin, _aMax, -_jMax);
  IF validProfileCounter >= 0
  THEN
    Get := CalculateBlock(block);
    RETURN;
	END_IF  
END_IF

Get := CalculateBlock(block);
END_METHOD

METHOD PRIVATE RemoveProfile : BOOL
VAR_INPUT
  index : INT;
END_VAR
VAR
  i : INT;
END_VAR
// todo, this is pretty slow in twincat
FOR i:=index TO validProfileCounter-2
DO
  validProfiles[i] := validProfiles[i + 1];
END_FOR

validProfileCounter := validProfileCounter - 1;
END_METHOD

METHOD Set
VAR_INPUT
  p0, v0, a0 : LREAL;
  pf, vf, af : LREAL;
  vMax, vMin : LREAL;
  aMax, aMin : LREAL;
  jMax : LREAL;  
END_VAR
THIS^.p0 := p0;
THIS^.v0 := v0;
THIS^.a0 := a0;
THIS^.pf := pf;
THIS^.vf := vf;
THIS^.af := af;
_vMax := vMax;
_vMin := vMin;
_aMax := aMax;
_aMin := aMin;
_jMax := jMax;

pd := pf - p0;

v0_v0 := v0 * v0;
vf_vf := vf * vf;

a0_a0 := a0 * a0;
af_af := af * af;

a0_p3 := a0 * a0_a0;
a0_p4 := a0_a0 * a0_a0;
af_p3 := af * af_af;
af_p4 := af_af * af_af;

// max values needs to be invariant to plus minus sign change
jMax_jMax := jMax * jMax;
END_METHOD

METHOD PRIVATE time_acc0
VAR_INPUT
  Profile : REFERENCE TO ProfileDesc;
  vMax, vMin, aMax, aMin, jMax : LREAL;
END_VAR
h3 := (a0_a0 - af_af)/(2*aMax*jMax) + (vf - v0)/aMax;
t_max := (aMax - aMin)/jMax;

h0 := 3*(af_p4 - a0_p4) + 8*(a0_p3 - af_p3)*aMax + 24*aMax*jMax*(af*vf - a0*v0) - 6*a0_a0*(aMax*aMax - 2*jMax*v0) + 6*af_af*(aMax*aMax - 2*jMax*vf) + 12*jMax*(jMax*(vf_vf - v0_v0 - 2*aMax*pd) - aMax*aMax*(vf - v0));
h2 := -af_af + aMax*aMax + 2*jMax*vf;
    
polynom[1] := (-2*aMax)/jMax;
polynom[2] := h2/jMax_jMax;
polynom[3] := 0;
polynom[4] := h0/(12*jMax_jMax*jMax_jMax);

t_min := (aMax - af)/jMax;
    
Roots.SolveQuartMonic(ADR(polynom[1]), 4, rootCount:=rootCount, roots:=root);
FOR i:=0 TO rootCount
DO
  t := root[i];
  IF t < t_min OR_ELSE t > t_max
  THEN
    CONTINUE;
  END_IF
  
  // Single Newton step (regarding pd)
  IF t > Constants.DoubleEpsilon
  THEN
    h1 := jMax*t;
    orig := h0/(24*aMax*jMax_jMax) + t*t*(h2 + h1*(h1 - 2*aMax))/(2*aMax);
    deriv := t*(h2 + h1*(2*h1 - 3*aMax))/aMax;
    IF ABS(deriv) > Constants.DoubleEpsilon
    THEN
      t := t - orig / deriv;
    END_IF
  END_IF
  
  IF ABS(deriv) < Constants.DoubleEpsilon
  THEN
    CONTINUE;
	END_IF
  
  Profile.t[0] := (-a0 + aMax)/jMax;
  Profile.t[1] := h3 - 2*t + jMax/aMax*t*t;
  Profile.t[2] := t;
  Profile.t[3] := 0;
  Profile.t[4] := 0;
  Profile.t[5] := 0;
  Profile.t[6] := (af - aMax)/jMax + t;
  
  IF (Profile.CheckVel(ProfileJerkSigns.Uddu, ProfileLimits.Acc0, jMax, vMax, vMin, aMax, aMin, setLimits:=FALSE))
  THEN
    AddProfile(Profile, jMax);        
  END_IF
END_FOR
END_METHOD

METHOD PRIVATE time_acc0_acc1
VAR_INPUT
  Profile : REFERENCE TO ProfileDesc;
  vMax, vMin, aMax, aMin, jMax : LREAL;
END_VAR
VAR
  temp : LREAL;
END_VAR
h1 := (3*(af_p4*aMax - a0_p4*aMin) + aMax*aMin*(8*(a0_p3 - af_p3) + 3*aMax*aMin*(aMax - aMin) + 6*aMin*af_af - 6*aMax*a0_a0) + 12*jMax*(aMax*aMin*((aMax - 2*a0)*v0 - (aMin - 2*af)*vf) + aMin*a0_a0*v0 - aMax*af_af*vf))/(3*(aMax - aMin)*jMax_jMax) + 4*(aMax*vf_vf - aMin*v0_v0 - 2*aMin*aMax*pd)/(aMax - aMin);
IF (h1 >= 0) // check if h1 isNan
THEN
  h1 := SQRT(h1) * 0.5;
  h2 := a0_a0/(2*aMax*jMax) + (aMin - 2*aMax)/(2*jMax) - v0/aMax;
  h3 := -af_af/(2*aMin*jMax) - (aMax - 2*aMin)/(2*jMax) + vf/aMin;
  
  // UDDU: Solution 2
  IF h2 > h1/aMax AND_THEN h3 > -h1/aMin
  THEN
    profile.t[0] := (-a0 + aMax)/jMax;
    profile.t[1] := h2 - h1/aMax;
    profile.t[2] := aMax/jMax;
    profile.t[3] := 0;
    profile.t[4] := -aMin/jMax;
    profile.t[5] := h3 + h1/aMin;
    profile.t[6] := profile.t[4] + af/jMax;
  
    IF (Profile.CheckVel(ProfileJerkSigns.Uddu, ProfileLimits.Acc0Acc1, jMax, vMax, vMin, aMax, aMin, setLimits:=TRUE))
    THEN
      AddProfile(Profile, jMax);            
    END_IF
  END_IF
  
  // UDDU: Solution 1  
  IF h2 > -h1/aMax AND_THEN h3 > h1/aMin
  THEN
    Profile.t[0] := (-a0 + aMax)/jMax;
    Profile.t[1] := h2 + h1/aMax;
    Profile.t[2] := aMax/jMax;
    Profile.t[3] := 0;
    Profile.t[4] := -aMin/jMax;
    Profile.t[5] := h3 - h1/aMin;
    Profile.t[6] := Profile.t[4] + af/jMax;
  
    IF (Profile.CheckVel(ProfileJerkSigns.Uddu, ProfileLimits.Acc0Acc1, jMax, vMax, vMin, aMax, aMin, setLimits:=TRUE))
    THEN
      AddProfile(Profile, jMax);              
    END_IF
	END_IF  
END_IF
END_METHOD

METHOD PRIVATE time_acc0_two_step
VAR_INPUT
  Profile : REFERENCE TO ProfileDesc;
  vMax, vMin, aMax, aMin, jMax : LREAL;
END_VAR
IF ABS(2*a0*jMax) > Constants.Epsilon
THEN
  // Two step
  Profile.t[0] := 0;
  Profile.t[1] := (af_af - a0_a0 + 2*jMax*(vf - v0))/(2*a0*jMax);
  Profile.t[2] := (a0 - af)/jMax;
  Profile.t[3] := 0;
  Profile.t[4] := 0;
  Profile.t[5] := 0;
  Profile.t[6] := 0;
  
  IF (Profile.CheckVel(ProfileJerkSigns.Uddu, ProfileLimits.Acc0, jMax, vMax, vMin, aMax, aMin, setLimits:=FALSE))
  THEN
    AddProfile(Profile, jMax);
    RETURN;
  END_IF
END_IF

// Three step - Removed pf
Profile.t[0] := (-a0 + aMax)/jMax;
Profile.t[1] := (a0_a0 + af_af - 2*aMax*aMax + 2*jMax*(vf - v0))/(2*aMax*jMax);
Profile.t[2] := (-af + aMax)/jMax;
Profile.t[3] := 0;
Profile.t[4] := 0;
Profile.t[5] := 0;
Profile.t[6] := 0;

IF (Profile.CheckVel(ProfileJerkSigns.Uddu, ProfileLimits.Acc0, jMax, vMax, vMin, aMax, aMin, setLimits:=FALSE))
THEN
  AddProfile(Profile, jMax);
  RETURN;     
END_IF


// Three step - Removed aMax
h0 := 3*(af_af - a0_a0 + 2*jMax*(v0 + vf));
h2 := a0_p3 + 2*af_p3 + 6*jMax_jMax*pd + 6*(af - a0)*jMax*vf - 3*a0*af_af;
h1 := 2*(2*h2*h2 + h0*(a0_p4 - 6*a0_a0*(af_af + 2*jMax*vf) + 8*a0*(af_p3 + 3*jMax_jMax*pd + 3*af*jMax*vf) - 3*(af_p4 + 4*af_af*jMax*vf + 4*jMax_jMax*(vf_vf - v0_v0))));
IF h1 >= 0 AND_THEN ABS(h0) > Constants.DoubleEpsilon
THEN
  h1 := SQRT(h1) * ABS(jMax) / jMax;
  
  Profile.t[0] := (4*af_p3 + 2*a0_p3 - 6*a0*af_af + 12*jMax_jMax*pd + 12*(af - a0)*jMax*vf + h1)/(2*jMax*h0);
  Profile.t[1] := -h1/(jMax*h0);
  Profile.t[2] := (-4*a0_p3 - 2*af_p3 + 6*a0_a0*af + 12*jMax_jMax*pd - 12*(af - a0)*jMax*v0 + h1)/(2*jMax*h0);
  Profile.t[3] := 0;
  Profile.t[4] := 0;
  Profile.t[5] := 0;
  Profile.t[6] := 0;
  
  IF (Profile.CheckVel(ProfileJerkSigns.Uddu, ProfileLimits.Acc0, jMax, vMax, vMin, aMax, aMin, setLimits:=FALSE))
  THEN
    AddProfile(Profile, jMax);
    RETURN;     
  END_IF
END_IF
END_METHOD

METHOD PRIVATE time_acc1
VAR_INPUT
  Profile : REFERENCE TO ProfileDesc;
  vMax, vMin, aMax, aMin, jMax : LREAL;
END_VAR
h3 := -(a0_a0 + af_af)/(2*jMax*aMin) + aMin/jMax + (vf - v0)/aMin;
t_max := (-a0 + aMax)/jMax;

h0 := 3*(a0_p4 - af_p4) + 8*(af_p3 - a0_p3)*aMin + 6*(a0_a0 - af_af)*aMin*aMin + 12*jMax*(af_af*vf + a0_a0*v0 + 2*aMin*(jMax*pd - a0*v0 - af*vf) + aMin*aMin*(v0 + vf) + jMax*(v0_v0 - vf_vf));
h2 := a0_a0 - a0*aMin + 2*jMax*v0;

polynom[0] := 1.0;
polynom[1] := (2*(2*a0 - aMin))/jMax;
polynom[2] := (5*a0_a0 + aMin*(aMin - 6*a0) + 2*jMax*v0)/jMax_jMax;
polynom[3] := 2*(a0 - aMin)*h2/(jMax_jMax*jMax);
polynom[4] := h0/(12*jMax_jMax*jMax_jMax);

t_min := -(a0 - aMin)/jMax;
    
Roots.SolveQuartMonic(ADR(polynom[1]), 4, rootCount:=rootCount, roots:=root);
FOR i:=0 TO rootCount
DO
  t := root[i];
  IF (t < t_min OR_ELSE t > t_max) THEN
    CONTINUE;
  END_IF 

  IF t > Constants.DoubleEpsilon
  THEN
    // Double Newton step (regarding pd)
    h1 := jMax*t*t;
    orig := -(h0 + 12*jMax*(2*a0_p3*t + 2*a0*(aMin - 2*jMax*t)*(aMin*t - h1) + 4*jMax*t*a0*v0 + a0_a0*(-4*aMin*t + 5*h1) + aMin*aMin*h1 + jMax*(h1 - 2*aMin*t)*(h1 + 2*v0)))/(24*aMin*jMax_jMax);
    deriv := -((a0 - aMin + jMax*t)*(h2 + jMax*((4*a0 - aMin)*t + 2*h1)))/(aMin*jMax);
            
    IF ABS(deriv) > Constants.DoubleEpsilon
    THEN
      t := t - MIN(orig / deriv, t);
      
      h1 := jMax*t*t;
      orig := -(h0 + 12*jMax*(2*a0_p3*t + 2*a0*(aMin - 2*jMax*t)*(aMin*t - h1) + 4*jMax*t*a0*v0 + a0_a0*(-4*aMin*t + 5*h1) + aMin*aMin*h1 + jMax*(h1 - 2*aMin*t)*(h1 + 2*v0)))/(24*aMin*jMax_jMax);
      IF (ABS(orig) > 1E-9)
      THEN
        deriv := -((a0 - aMin + jMax*t)*(h2 + jMax*((4*a0 - aMin)*t + 2*h1)))/(aMin*jMax);
        
        IF ABS(deriv) > Constants.DoubleEpsilon
        THEN
          t := t - orig / deriv; 
        END_IF
      END_IF 
    END_IF  
	END_IF

  Profile.t[0] := t;
  Profile.t[1] := 0;
  Profile.t[2] := (a0 - aMin)/jMax + t;
  Profile.t[3] := 0;
  Profile.t[4] := 0;
  Profile.t[5] :=  h3 - 2*a0/aMin*t - jMax/aMin*t*t;
  Profile.t[6] := (af - aMin)/jMax;
  
  IF (Profile.CheckVel(ProfileJerkSigns.Uddu, ProfileLimits.Acc1, jMax, vMax, vMin, aMax, aMin, setLimits:=TRUE))
  THEN
    AddProfile(Profile, jMax);
  END_IF
END_FOR
END_METHOD

METHOD PRIVATE time_acc1_vel_two_step
VAR_INPUT
  Profile : REFERENCE TO ProfileDesc;
  vMax, vMin, aMax, aMin, jMax : LREAL;
END_VAR
profile.t[0] := 0;
profile.t[1] := 0;
profile.t[2] := a0/jMax;
profile.t[3] := -(3*af_p4 - 8*aMin*(af_p3 - a0_p3) - 24*aMin*jMax*(a0*v0 - af*vf) + 6*af_af*(aMin*aMin - 2*jMax*vf) - 12*jMax*(2*aMin*jMax*pd + aMin*aMin*(vf + vMax) + jMax*(vMax*vMax - vf_vf) + aMin*a0*(a0_a0 - 2*jMax*(v0 + vMax))/jMax))/(24*aMin*jMax_jMax*vMax);
profile.t[4] := -aMin/jMax;
profile.t[5] := -(af_af/2 - aMin*aMin + jMax*(vMax - vf))/(aMin*jMax);
profile.t[6] := profile.t[4] + af/jMax;

IF (Profile.CheckVel(ProfileJerkSigns.Uddu, ProfileLimits.Acc1Vel, jMax, vMax, vMin, aMax, aMin, setLimits:=FALSE))
THEN
  AddProfile(Profile, jMax);
  RETURN;        
END_IF
END_METHOD

METHOD PRIVATE time_all_vel
VAR_INPUT
  Profile : REFERENCE TO ProfileDesc;
  vMax, vMin, aMax, aMin, jMax : LREAL;
END_VAR
// ACC0_ACC1_VEL
Profile.t[0] := (-a0 + aMax)/jMax;
Profile.t[1] := (a0_a0*0.5 - aMax*aMax - jMax*(v0 - vMax))/(aMax*jMax);
Profile.t[2] := aMax/jMax;
Profile.t[3] := (3*(a0_p4*aMin - af_p4*aMax) + 8*aMax*aMin*(af_p3 - a0_p3 + 3*jMax*(a0*v0 - af*vf)) + 6*a0_a0*aMin*(aMax*aMax - 2*jMax*v0) - 6*af_af*aMax*(aMin*aMin - 2*jMax*vf) - 12*jMax*(aMax*aMin*(aMax*(v0 + vMax) - aMin*(vf + vMax) - 2*jMax*pd) + (aMin - aMax)*jMax*vMax*vMax + jMax*(aMax*vf_vf - aMin*v0_v0)))/(24*aMax*aMin*jMax_jMax*vMax);
Profile.t[4] := -aMin/jMax;
Profile.t[5] := -(af_af*0.5 - aMin*aMin - jMax*(vf - vMax))/(aMin*jMax);
Profile.t[6] := Profile.t[4] + af/jMax;

IF (Profile.CheckVel(ProfileJerkSigns.Uddu, ProfileLimits.Acc0Acc1Vel, jMax, vMax, vMin, aMax, aMin, setLimits:=FALSE))
THEN
  AddProfile(Profile, jMax);
  RETURN;    
END_IF

// ACC1_VEL
t_acc0  := a0_a0/(2*jMax_jMax) + (vMax - v0)/jMax;
IF t_acc0 >= 0
THEN
  t_acc0 := SQRT(t_acc0 );
  Profile.t[0] := t_acc0  - a0/jMax;
  Profile.t[1] := 0;
  Profile.t[2] := t_acc0 ;
  Profile.t[3] := -(3*af_p4 - 8*aMin*(af_p3 - a0_p3) - 24*aMin*jMax*(a0*v0 - af*vf) + 6*af_af*(aMin*aMin - 2*jMax*vf) - 12*jMax*(2*aMin*jMax*pd + aMin*aMin*(vf + vMax) + jMax*(vMax*vMax - vf_vf) + aMin*t_acc0 *(a0_a0 - 2*jMax*(v0 + vMax))))/(24*aMin*jMax_jMax*vMax);
  //Profile.t[4] := -aMin/jMax;
  //Profile.t[5] := -(af_af*0.5 - aMin*aMin + jMax*(vMax - vf))/(aMin*jMax);
  //Profile.t[6] := Profile.t[4] + af/jMax;
        
  IF (Profile.CheckVel(ProfileJerkSigns.Uddu, ProfileLimits.Acc1Vel, jMax, vMax, vMin, aMax, aMin, setLimits:=FALSE)) 
  THEN
    AddProfile(Profile, jMax); 
    RETURN; 
  END_IF
END_IF

// ACC0_VEL
t_acc1 := 0.5*af_af/(jMax_jMax) + (vMax - vf)/jMax;
IF t_acc1 >= 0
THEN
  t_acc1 := SQRT(t_acc1);
  Profile.t[0] := (-a0 + aMax)/jMax;
  Profile.t[1] := (a0_a0*0.5 - aMax*aMax - jMax*(v0 - vMax))/(aMax*jMax);
  Profile.t[2] := aMax/jMax;
  Profile.t[3] := (3*a0_p4 + 8*(af_p3 - a0_p3)*aMax + 24*aMax*jMax*(a0*v0 - af*vf) + 6*a0_a0*(aMax*aMax - 2*jMax*v0) - 12*jMax*(-2*aMax*jMax*pd + aMax*aMax*(v0 + vMax) + jMax*(vMax*vMax - v0_v0) + (2*(vf + vMax)*jMax - af_af)*aMax*t_acc1))/(24*aMax*jMax_jMax*vMax);
  Profile.t[4] := t_acc1;
  Profile.t[5] := 0;
  Profile.t[6] := t_acc1 + af/jMax;
  
  IF (Profile.CheckVel(ProfileJerkSigns.Uddu, ProfileLimits.Acc0Vel, jMax, vMax, vMin, aMax, aMin, setLimits:=FALSE)) 
  THEN
    AddProfile(Profile, jMax);
    RETURN;
  END_IF
END_IF

// VEL
// Solution 3/4
IF t_acc0 >= 0 AND_THEN t_acc1 >= 0
THEN
  Profile.t[0] := t_acc0 - a0/jMax;
  Profile.t[1] := 0;
  Profile.t[2] := t_acc0;
  Profile.t[3] := (af_p3 - a0_p3)/(3.0*jMax_jMax*vMax) + (a0*v0 - af*vf + (af_af*t_acc1 + a0_a0*t_acc0)*0.5)/(jMax*vMax) - (v0/vMax + 1.0)*t_acc0 - (vf/vMax + 1.0)*t_acc1 + pd/vMax;
  //Profile.t[4] := t_acc1;
  //Profile.t[5] := 0;
  //Profile.t[6] := t_acc1 + af/jMax;
  
  IF (Profile.CheckVel(ProfileJerkSigns.Uddu, ProfileLimits.Vel, jMax, vMax, vMin, aMax, aMin, setLimits:=FALSE))
  THEN
    AddProfile(Profile, jMax);
    RETURN;
  END_IF
END_IF
END_METHOD

METHOD PRIVATE time_none
VAR_INPUT
  Profile : REFERENCE TO ProfileDesc;  
  vMax : LREAL;
  vMin : LREAL;  
  aMax : LREAL;
  aMin : LREAL;
  jMax : LREAL;
END_VAR
// UDDU
IF (ABS(v0) < Constants.DoubleEpsilon AND_THEN ABS(a0) < Constants.DoubleEpsilon AND_THEN ABS(vf) < Constants.DoubleEpsilon AND_THEN ABS(af) < Constants.DoubleEpsilon)
THEN
  Profile.t[0] := Cbrt(pd/(2*jMax));
  Profile.t[1] := 0;
  Profile.t[2] := 2*Profile.t[0];
  Profile.t[3] := 0;
  Profile.t[4] := 0;
  Profile.t[5] := 0;
  Profile.t[6] := Profile.t[0];
  
  IF (Profile.CheckVel(ProfileJerkSigns.Uddu, ProfileLimits.None, jMax, vMax, vMin, aMax, aMin, setLimits:=FALSE))
  THEN
    AddProfile(Profile, jMax); 
  END_IF
  
  RETURN; 
END_IF

        
IF (ABS(a0 - af) < Constants.DoubleEpsilon AND_THEN ABS(v0 + vf) < Constants.DoubleEpsilon AND_THEN ABS(p0 - pf) < Constants.DoubleEpsilon) 
THEN
  h1 := SQRT(a0_a0 - 2*jMax*v0);

  // Solution 3
  Profile.t[0] := -(a0 + h1)/jMax;
  Profile.t[1] := 0;
  Profile.t[2] := Profile.t[0];
  Profile.t[3] := 0;
  Profile.t[4] := 0;
  Profile.t[5] := 0;
  Profile.t[6] := 0;

  IF (Profile.CheckVel(ProfileJerkSigns.Uddu, ProfileLimits.None, jMax, vMax, vMin, aMax, aMin, setLimits:=FALSE))
  THEN
    AddProfile(Profile, jMax);                
  END_IF
        
  // Solution 4
  Profile.t[0] := -(a0 - h1)/jMax;
  Profile.t[1] := 0;
  Profile.t[2] := Profile.t[0];
  Profile.t[3] := 0;
  Profile.t[4] := 0;
  Profile.t[5] := 0;
  Profile.t[6] := 0;

  IF (Profile.CheckVel(ProfileJerkSigns.Uddu, ProfileLimits.None, jMax, vMax, vMin, aMax, aMin, setLimits:=FALSE))
  THEN
    AddProfile(Profile, jMax);                
  END_IF
        
  RETURN;        
END_IF

// UDDU / UDUD modern, this one is in particular prone to numerical issues
// UDUD Strategy: t7 == 0 (equals UDDU)
h2 := (a0_a0 - af_af)/(2*jMax) + (vf - v0);
h2_h2 := h2*h2;
polynom[1] := 0.0;
polynom[2] := (-2*(a0_a0 + af_af - 2*jMax*(v0 + vf)))/jMax_jMax;
polynom[3] := 4*(a0_p3 - af_p3 + 3*jMax*(af*vf - a0*v0))/(3*jMax*jMax_jMax) - 4*pd/jMax;
polynom[4] := -h2_h2/jMax_jMax;

t_min := (a0 - af)/jMax;
t_max := (aMax - aMin)/jMax;
        
Roots.SolveQuartMonic(ADR(polynom[1]), 4, rootCount:=rootCount, roots:=root);
FOR i:=0 TO rootCount
DO
  t := root[i];
  IF t < t_min OR_ELSE t > t_max
  THEN
    CONTINUE;
	END_IF
            
  // Single Newton-step (regarding pd)
  IF (t > Constants.DoubleEpsilon)
  THEN
    h1 := jMax*t*t;    
    orig := -h2_h2/(4*jMax*t) + h2*(af/jMax + t) + (4*a0_p3 + 2*af_p3 - 6*a0_a0*(af + 2*jMax*t) + 12*(af - a0)*jMax*v0 + 3*jMax_jMax*(-4*pd + (h1 + 8*v0)*t))/(12*jMax_jMax);
    deriv := h2 + 2*v0 - a0_a0/jMax + h2_h2/(4*h1) + (3*h1)/4;
    IF ABS(deriv) < Constants.DoubleEpsilon
    THEN
      CONTINUE;
    END_IF
    
    t := t - orig / deriv;
  END_IF
  
  IF (t <= Constants.DoubleEpsilon)
  THEN
    CONTINUE;
  END_IF
  
  h0 := h2/(2*jMax*t);
  Profile.t[0] := h0 + t*0.5 - a0/jMax;
  Profile.t[1] := 0;
  Profile.t[2] := t;
  Profile.t[3] := 0;
  Profile.t[4] := 0;
  Profile.t[5] := 0;
  Profile.t[6] := -h0 + t*0.5 + af/jMax;

  IF (Profile.CheckVel(ProfileJerkSigns.Uddu, ProfileLimits.None, jMax, vMax, vMin, aMax, aMin, setLimits:=FALSE)) 
  THEN
    AddProfile(Profile, jMax);            
  END_IF
  
END_FOR
END_METHOD

METHOD PRIVATE time_none_two_step
VAR_INPUT
  Profile : REFERENCE TO ProfileDesc;
  vMax, vMin, aMax, aMin, jMax : LREAL;
END_VAR
// Two step
{}
  h0 := (a0_a0 + af_af)/2 + jMax*(vf - v0);
  IF h0 >= 0
  THEN
    h0 := SQRT(h0) * ABS(jMax) / jMax;
    profile.t[0] := (h0 - a0)/jMax;
    profile.t[1] := 0;
    profile.t[2] := (h0 - af)/jMax;
    profile.t[3] := 0;
    profile.t[4] := 0;
    profile.t[5] := 0;
    profile.t[6] := 0;
    
    IF (profile.CheckVel(ProfileJerkSigns.Uddu, ProfileLimits.None, jMax, vMax, vMin, aMax, aMin, setLimits:=FALSE))
    THEN 
      AddProfile(profile, jMax);
      RETURN;
    END_IF
	END_IF
{}
  
  // Single step
{}
  profile.t[0] := (af - a0)/jMax;
  profile.t[1] := 0;
  profile.t[2] := 0;
  profile.t[3] := 0;
  profile.t[4] := 0;
  profile.t[5] := 0;
  profile.t[6] := 0;
  
  IF (profile.CheckVel(ProfileJerkSigns.Uddu, ProfileLimits.None, jMax, vMax, vMin, aMax, aMin, setLimits:=FALSE))
  THEN 
    AddProfile(profile, jMax);
    RETURN;
  END_IF
{}
END_METHOD

METHOD PRIVATE time_vel_two_step
VAR_INPUT
  Profile : REFERENCE TO ProfileDesc;
  vMax, vMin, aMax, aMin, jMax : LREAL;
END_VAR
h1 := af_af/(2*jMax_jMax) + (vMax - vf)/jMax;

IF h1 >= 0
THEN
  h1 := SQRT(h1);
  
  // Four step
  {}    
    // Solution 3/4
    profile.t[0] := -a0/jMax;
    profile.t[1] := 0;
    profile.t[2] := 0;
    profile.t[3] := (af_p3 - a0_p3)/(3*jMax_jMax*vMax) + (a0*v0 - af*vf + (af_af*h1)/2)/(jMax*vMax) - (vf/vMax + 1.0)*h1 + pd/vMax;
    profile.t[4] := h1;
    profile.t[5] := 0;
    profile.t[6] := h1 + af/jMax;
  
    IF Profile.CheckVel(ProfileJerkSigns.Uddu, ProfileLimits.Vel, jMax, vMax, vMin, aMax, aMin, setLimits:=FALSE)
    THEN
      addProfile(profile, jMax);
      RETURN;
    END_IF 
  {}
  
  {}    
    // Four step        
    Profile.t[0] := 0;
    Profile.t[1] := 0;
    Profile.t[2] := a0/jMax;
    Profile.t[3] := (af_p3 - a0_p3)/(3.0*jMax_jMax*vMax) + (a0*v0 - af*vf + (af_af*h1 + a0_p3/jMax)*0.5)/(jMax*vMax) - (v0/vMax + 1.0)*a0/jMax - (vf/vMax + 1.0)*h1 + pd/vMax;
    Profile.t[4] := h1;
    Profile.t[5] := 0;
    Profile.t[6] := h1 + af/jMax;
    
    IF (Profile.CheckVel(ProfileJerkSigns.Uddu, ProfileLimits.Vel, jMax, vMax, vMin, aMax, aMin, setLimits:=FALSE))
    THEN
      AddProfile(Profile, jMax); 
      RETURN;       
    END_IF
  {}
END_IF
END_METHOD

END_FUNCTION_BLOCK

// ---- Struckig/Profile/ProfileDesc.TcPOU
/// The state Profile for position, velocity, acceleration and jerk for a single DoF
FUNCTION_BLOCK INTERNAL ProfileDesc
VAR_INPUT
  Limits : ProfileLimits;
  Direction : ProfileDirection;
  JerkSigns : ProfileJerkSigns;
  
  t, t_sum, j : ARRAY[0..6] OF LREAL;
  a, v, p : ARRAY[0..7] OF LREAL;

  pf, vf, af : LREAL; // Target (final) kinematic state
  
  hasBrake : BOOL;
  t_brake : LREAL; // Total time of the braking segments
  t_brakes, j_brakes, a_brakes, v_brakes, p_brakes : ARRAY[0..1] OF LREAL; // Allow up to two segments of braking before the "correct" Profile starts 
END_VAR

/// For velocity interface
METHOD CheckForVelocity : BOOL
VAR_INPUT
  jerkSigns : ProfileJerkSigns;
  limits : ProfileLimits;  
  jf : LREAL;
  aMax : LREAL;
  aMin : LREAL;  
END_VAR
VAR
  i : INT;
  aUppLim : LREAL;
  aLowLim : LREAL;
END_VAR
IF (t[0] < 0)
THEN
  RETURN;
END_IF

t_sum[0] := t[0];
FOR i:=0 TO 5
DO
  IF (t[i+1] < 0)
  THEN
    RETURN;
  END_IF
  
  t_sum[i+1] := t_sum[i] + t[i+1];
END_FOR


IF limits = ProfileLimits.Acc0
THEN
  IF t[1] < Constants.Epsilon
  THEN
    RETURN;
  END_IF
END_IF


IF (t_sum[6] > 1E12) { // For numerical reasons, is that needed?}
THEN
  RETURN;        
END_IF

IF jerkSigns = ProfileJerkSigns.Uddu
THEN
  j[0] := jf;
  j[1] := 0;
  j[2] := -jf;
  j[3] := 0;
  j[4] := -jf;
  j[5] := 0;
  j[6] := jf;          
ELSE
  j[0] := jf;
  j[1] := 0;
  j[2] := -jf;
  j[3] := 0;
  j[4] := jf;
  j[5] := 0;
  j[6] := -jf;
END_IF


FOR i:=0 TO 6
DO
  a[i+1] := a[i] + t[i] * j[i];
  v[i+1] := v[i] + t[i] * (a[i] + t[i] * j[i] / 2);
  p[i+1] := p[i] + t[i] * (v[i] + t[i] * (a[i] / 2 + t[i] * j[i] / 6));        
END_FOR

      
THIS^.JerkSigns := jerkSigns;
THIS^.Limits := limits;

aUppLim := SEL((aMax > 0), aMin, aMax) + 5E-12;
aLowLim := SEL((aMax > 0), aMax, aMin) - 5E-12;

// Velocity limit can be broken in the beginning if both initial velocity and acceleration are too high
CheckForVelocity := ABS(v[7] - vf) < 1E-8
    AND_THEN ABS(a[7] - af) < 1E-10 // This is not really needed, but we want to double check
    AND_THEN a[1] >= aLowLim AND_THEN a[3] >= aLowLim AND_THEN a[5] >= aLowLim
    AND_THEN a[1] <= aUppLim AND_THEN a[3] <= aUppLim AND_THEN a[5] <= aUppLim;
END_METHOD

/// For velocity interface
METHOD CheckForVelocityWithTiming : BOOL
VAR_INPUT
  jerkSigns : ProfileJerkSigns;
  limits : ProfileLimits;  
  jf : LREAL;
  aMax : LREAL;
  aMin : LREAL;  
END_VAR
VAR
  i : INT;
  aUppLim : LREAL;
  aLowLim : LREAL;
END_VAR
// Time doesn't need to be checked as every profile has a: tf - ... equation
CheckForVelocityWithTiming := CheckForVelocity(jerkSigns, limits, jf, aMax, aMin);
END_METHOD

METHOD CheckPositionExtremum : BOOL
VAR_INPUT
  t_ext, t_sum, t, p, v, a, j : LREAL;
END_VAR
VAR_IN_OUT
  ext : PositionExtremaDesc;     
END_VAR
VAR
  p_ext, v_Ext, a_ext : LREAL;
END_VAR
IF (0 < t_ext AND_THEN t_ext < t)
THEN
  Integrate(t_ext, p, v, a, j, p:=p_ext, v:=v_ext, a:=a_ext);
  IF (a_ext > 0 AND_THEN p_ext < ext.Minimum)
  THEN
    ext.Minimum := p_ext;
    ext.Tmin := t_sum + t_ext;
   ELSIF (a_ext < 0 AND_THEN p_ext > ext.Maximum) 
   THEN
    ext.Maximum := p_ext;
    ext.Tmax := t_sum + t_ext; 
  END_IF
END_IF
END_METHOD

METHOD CheckStepForPositionExtremum : BOOL
VAR_INPUT
  t_sum, t, p, v, a, j : LREAL;
END_VAR
VAR_IN_OUT
  ext : PositionExtremaDesc;  
END_VAR
VAR
  d, d_sqrt : LREAL;
END_VAR
IF (p < ext.Minimum)
THEN 
  ext.Minimum := p;
  ext.Tmin := t_sum;
END_IF

IF (p > ext.Maximum)
THEN 
  ext.Maximum := p;
  ext.Tmax := t_sum;
END_IF

IF (j <> 0) 
THEN
  d := a * a - 2 * j * v;
  IF (ABS(d) < Constants.DoubleEpsilon)
  THEN
    CheckPositionExtremum(-a / j, t_sum, t, p, v, a, j, ext:=ext);
   ELSIF (d > 0) 
   THEN
    d_sqrt := SQRT(d);
    CheckPositionExtremum((-a - D_sqrt) / j, t_sum, t, p, v, a, j, ext:=ext);
    CheckPositionExtremum((-a + D_sqrt) / j, t_sum, t, p, v, a, j, ext:=ext);           
  END_IF
END_IF
END_METHOD

/// For position interface
METHOD CheckVel : BOOL
VAR_INPUT
  jerkSigns : ProfileJerkSigns;    
  limits : ProfileLimits;
  jf : LREAL;
  vMax : LREAL;
  vMin : LREAL;  
  aMax : LREAL;
  aMin : LREAL;
  setLimits : BOOL;
END_VAR
VAR
  i : INT;
  v_a_zero : LREAL;
  vUppLim, vLowLim : LREAL;  
  aUppLim, aLowLim : LREAL;
END_VAR
IF (t[0] < 0) 
THEN
  RETURN;
END_IF

t_sum[0] := t[0];
FOR i:=0 TO 5
DO
  IF (t[i+1] < 0)
  THEN
    RETURN;
  END_IF
  
  t_sum[i+1] := t_sum[i] + t[i+1];  
END_FOR

IF limits = ProfileLimits.Acc0Acc1Vel OR_ELSE limits = ProfileLimits.Acc0Vel OR_ELSE limits = ProfileLimits.Acc1Vel OR_ELSE limits = ProfileLimits.Vel THEN
  IF (t[3] < Constants.Epsilon) 
  THEN
    RETURN;                    
  END_IF
END_IF

IF limits = ProfileLimits.Acc0 OR_ELSE limits = ProfileLimits.Acc0Acc1
THEN
  IF (t[1] < Constants.Epsilon) 
  THEN
    RETURN;                    
  END_IF
END_IF

IF limits = ProfileLimits.Acc1 OR_ELSE limits = ProfileLimits.Acc0Acc1
THEN
  IF (t[5] < Constants.Epsilon)
  THEN
    RETURN;            
  END_IF
END_IF

IF t_sum[6] > 1E12  // For numerical reasons, is that needed?
THEN
  RETURN;        
END_IF
        
IF jerkSigns = ProfileJerkSigns.Uddu
THEN
  j[0] := jf;
  j[1] := 0;
  j[2] := -jf;
  j[3] := 0;
  j[4] := -jf;
  j[5] := 0;
  j[6] := jf;
ELSE
  j[0] := jf;
  j[1] := 0;
  j[2] := -jf;
  j[3] := 0;
  j[4] := jf;
  j[5] := 0;
  j[6] := -jf;          
END_IF

vUppLim := SEL(vMax > 0, vMin, vMax) + 1E-12;
vLowLim := SEL(vMax > 0, vMax, vMin) - 1E-12;
        
FOR i:= 0 TO 6 
DO
  a[i+1] := a[i] + t[i] * j[i];
  v[i+1] := v[i] + t[i] * (a[i] + t[i] * j[i] / 2);
  p[i+1] := p[i] + t[i] * (v[i] + t[i] * (a[i] / 2 + t[i] * j[i] / 6));

  IF limits = ProfileLimits.Acc0Acc1Vel OR_ELSE limits = ProfileLimits.Acc0Acc1 OR_ELSE limits = ProfileLimits.Acc0Vel OR_ELSE limits = ProfileLimits.Acc1Vel OR_ELSE limits = ProfileLimits.Vel
  THEN
    IF i = 2
    THEN
     a[3] := 0.0;
    END_IF
  END_IF
  
  IF setLimits
  THEN
    IF limits = ProfileLimits.Acc1
    THEN
      IF i = 2
      THEN
        a[3] := aMin;
      END_IF
    ELSIF limits = ProfileLimits.Acc0Acc1
    THEN
      CASE i
      OF
      0: a[1] := aMax;
      4: a[5] := aMin;
      END_CASE  
    END_IF
  END_IF
  
  IF (i > 1 AND_THEN a[i+1] * a[i] < -Constants.Epsilon) 
  THEN
    v_a_zero := v[i] - (a[i] * a[i]) / (2 * j[i]);
    IF (v_a_zero > vUppLim OR_ELSE v_a_zero < vLowLim)
    THEN
      RETURN;        
		END_IF
  END_IF
END_FOR


THIS^.JerkSigns := jerkSigns;
THIS^.Limits := limits;

aUppLim := SEL(aMax > 0, aMin, aMax) + 1E-12;
aLowLim := SEL(aMax > 0, aMax, aMin) - 1E-12;

// Velocity limit can be broken in the beginning if both initial velocity and acceleration are too high
CheckVel := ABS(p[7] - pf) < 1E-8
    AND_THEN ABS(v[7] - vf) < 1E-8
    AND_THEN ABS(a[7] - af) < 1E-10 // This is not really needed, but we want to double check
    // AND_THEN ABS(v[3]) <= vMaxAbs AND_THEN ABS(v[4]) <= vMaxAbs AND_THEN ABS(v[5]) <= vMaxAbs AND_THEN ABS(v[6]) <= vMaxAbs
    AND_THEN a[1] >= aLowLim AND_THEN a[3] >= aLowLim AND_THEN a[5] >= aLowLim
    AND_THEN a[1] <= aUppLim AND_THEN a[3] <= aUppLim AND_THEN a[5] <= aUppLim
    AND_THEN v[3] <= vUppLim AND_THEN v[4] <= vUppLim AND_THEN v[5] <= vUppLim AND_THEN v[6] <= vUppLim
    AND_THEN v[3] >= vLowLim AND_THEN v[4] >= vLowLim AND_THEN v[5] >= vLowLim AND_THEN v[6] >= vLowLim; // this is not really needed, but we want to double check
END_METHOD

METHOD CheckWithTiming : BOOL
VAR_INPUT
  jerkSigns : ProfileJerkSigns;    
  limits : ProfileLimits;
  tf : LREAL;
  jf : LREAL;
  vMax : LREAL;
  vMin : LREAL;  
  aMax : LREAL;
  aMin : LREAL;  
END_VAR
// Time doesn't need to be checked as every Profile has a: tf - ... equation
CheckWithTiming := CheckVel(jerkSigns, limits, jf, vMax, vMin, aMax, aMin, setLimits:=FALSE); // && (std::abs(t_sum[6] - tf) < 1e-8)
END_METHOD

METHOD CheckWithTiming2 : BOOL
VAR_INPUT
  jerkSigns : ProfileJerkSigns;    
  limits : ProfileLimits;
  tf : LREAL;
  jf : LREAL;
  vMax : LREAL;
  vMin : LREAL;  
  aMax : LREAL;
  aMin : LREAL;
  jMax  : LREAL;
END_VAR
CheckWithTiming2 := (ABS(jf) < ABS(jMax) + 1e-12) AND_THEN CheckWithTiming(jerkSigns, limits, tf, jf, vMax, vMin, aMax, aMin);
END_METHOD

METHOD FirstStateAtPosition : BOOL
VAR_INPUT
  pt, offset : LREAL;
END_VAR
VAR_IN_OUT
  t_t, v_t, a_t : LREAL;
END_VAR
VAR
  i,h : INT;
  p_t : LREAL;
  polynom : ARRAY[0..4] OF LREAL;
  rootCount : INT;
  root : ARRAY[0..6] OF LREAL;
END_VAR
FOR i:=0 TO 6
DO
  IF ABS(p[i] - pt) < Constants.Epsilon
  THEN
    t_t := offset + SEL(i>0, 0, t_sum[i-1]);
    v_t := v[i];
    a_t := a[i];
    FirstStateAtPosition := TRUE;
    RETURN;
	END_IF
  
  IF t[i] = 0
  THEN
    CONTINUE;
	END_IF
  
  polynom[0] := j[i]/6;
  polynom[1] := a[i]*0.5;
  polynom[2] := v[i];
  polynom[3] := p[i]-pt;
  Roots.SolveCub(ADR(polynom), rootCount:=rootCount, roots:=root);
  FOR h:=0 TO rootCount
  DO
    IF(0 < root[h] AND_THEN root[h] <= t[i])
    THEN
      t_t := offset + root[h] + SEL(i>0, 0, t_sum[i-1]);
      Integrate(root[h], p[i], v[i], a[i], j[i], p_t, v_t, a_t);
      FirstStateAtPosition := TRUE;
      RETURN;      
		END_IF
  END_FOR
  
END_FOR

IF ABS(pf-pt) < Constants.Epsilon
THEN
  t_t := offset + t_sum[6];
  v_t := vf;
  a_t := af;
  FirstStateAtPosition := TRUE;
  RETURN;      
END_IF
END_METHOD

 /// Integrate with constant jerk for duration t. Returns new position, new velocity, and new acceleration.
METHOD Integrate
VAR_INPUT
  t, p0, v0, a0, j  : LREAL;
END_VAR
VAR_IN_OUT
  p, v, a : LREAL;
END_VAR
p := p0 + t * (v0 + t * (a0 * 0.5 + t * j / 6));
v := v0 + t * (a0 + t * j * 0.5);
a := a0 + t * j;
END_METHOD

METHOD PositionExtrema : PositionExtremaDesc
VAR_INPUT
END_VAR
VAR
  i : INT;
  t_current_sum : LREAL;
END_VAR
PositionExtrema.Minimum := Constants.Infinity;
PositionExtrema.Maximum := -Constants.Infinity;

IF (hasBrake)
THEN
  IF (t_brakes[0] > 0.0)
  THEN
    CheckStepForPositionExtremum(0.0, t_brakes[0], p_brakes[0], v_brakes[0], a_brakes[0], j_brakes[0], PositionExtrema);
  
    IF (t_brakes[1] > 0.0) 
    THEN
      CheckStepForPositionExtremum(t_brakes[0], t_brakes[1], p_brakes[1], v_brakes[1], a_brakes[1], j_brakes[1], PositionExtrema);            
    END_IF
  END_IF
END_IF

t_current_sum := 0;        
FOR i:=0 TO 6
DO
  IF i > 0
  THEN
    t_current_sum := t_sum[i-1];
	END_IF
  
  CheckStepForPositionExtremum(t_current_sum + t_brakes[i], t[i], p[i], v[i], a[i], j[i], PositionExtrema);
END_FOR 

IF (pf < PositionExtrema.Minimum)
THEN
  PositionExtrema.Minimum := pf;
  PositionExtrema.Tmin := t_sum[6] + t_brakes[i];
END_IF 


IF (pf > PositionExtrema.Maximum) 
THEN
  PositionExtrema.Maximum := pf;
  PositionExtrema.Tmax := t_sum[6] + t_brakes[i];
END_IF
END_METHOD

/// Set boundary values for the position interface
METHOD SetBoundaryPosition
VAR_INPUT
  p0_new, v0_new, a0_new, pf_new, vf_new, af_new : LREAL;
END_VAR
a[0] := a0_new;
v[0] := v0_new;
p[0] := p0_new;
af := af_new;
vf := vf_new;
pf := pf_new;
END_METHOD

/// Set boundary values for the velocity interface
METHOD SetBoundaryVelocity
VAR_INPUT
  p0_new, v0_new, a0_new, vf_new, af_new : LREAL;
END_VAR
a[0] := a0_new;
v[0] := v0_new;
p[0] := p0_new;
af := af_new;
vf := vf_new;
END_METHOD

END_FUNCTION_BLOCK

// ---- Struckig/Position/PositionStep2.TcPOU
FUNCTION_BLOCK INTERNAL PositionStep2
VAR
  p0, v0, a0 : LREAL;
  tf, pf, vf, af : LREAL;
  _vMax, _vMin, _aMax, _aMin, _jMax : LREAL;
  
  // Pre-calculated expressions
  pd : LREAL;
  tf_tf, tf_p3, tf_p4 : LREAL;
  vd, vd_vd : LREAL;
  ad, ad_ad : LREAL;
  v0_v0, vf_vf : LREAL;
  a0_a0, a0_p3, a0_p4, a0_p5, a0_p6 : LREAL;
  af_af, af_p3, af_p4, af_p5, af_p6 : LREAL;
  jMax_jMax : LREAL;
  g1, g2 : LREAL;
  t_min, t_max : LREAL;
  up_first : BOOL;
  
  d_extremasCount : INT;
  d_extremas : ARRAY[0..6] OF LREAL;
  indices : ARRAY[0..6] OF INT;
END_VAR

METHOD Get : BOOL
VAR_INPUT
  Profile : REFERENCE TO ProfileDesc;
END_VAR
VAR_INST
  vMax, vMin, aMax, aMin, jMax : LREAL;
END_VAR
Profile.SetBoundaryPosition(p0, v0, a0, pf, vf, af);

up_first := (pd > tf * v0);
vMax := SEL(up_first, _vMin, _vMax);
vMin := SEL(up_first, _vMax, _vMin);
aMax := SEL(up_first, _aMin, _aMax);
aMin := SEL(up_first, _aMax, _aMin);
jMax := SEL(up_first, -_jMax, _jMax);

Get := time_acc0_acc1_vel(profile, vMax, vMin, aMax, aMin, jMax)
    OR_ELSE time_vel(profile, vMax, vMin, aMax, aMin, jMax)
    OR_ELSE time_acc0_vel(profile, vMax, vMin, aMax, aMin, jMax)
    OR_ELSE time_acc1_vel(profile, vMax, vMin, aMax, aMin, jMax)
    OR_ELSE time_acc0_acc1(profile, vMax, vMin, aMax, aMin, jMax)
    OR_ELSE time_acc0(profile, vMax, vMin, aMax, aMin, jMax)
    OR_ELSE time_acc1(profile, vMax, vMin, aMax, aMin, jMax)
    OR_ELSE time_none(profile, vMax, vMin, aMax, aMin, jMax)
    OR_ELSE time_acc0_acc1_vel(profile, vMin, vMax, aMin, aMax, -jMax)
    OR_ELSE time_vel(profile, vMin, vMax, aMin, aMax, -jMax)
    OR_ELSE time_acc0_vel(profile, vMin, vMax, aMin, aMax, -jMax)
    OR_ELSE time_acc1_vel(profile, vMin, vMax, aMin, aMax, -jMax)
    OR_ELSE time_acc0_acc1(profile, vMin, vMax, aMin, aMax, -jMax)
    OR_ELSE time_acc0(profile, vMin, vMax, aMin, aMax, -jMax)
    OR_ELSE time_acc1(profile, vMin, vMax, aMin, aMax, -jMax)
    OR_ELSE time_none(profile, vMin, vMax, aMin, aMax, -jMax);
END_METHOD

METHOD Set
VAR_INPUT
  tf : LREAL;
  p0, v0, a0 : LREAL;
  pf, vf, af : LREAL;
  vMax, vMin : LREAL;
  aMax, aMin : LREAL;
  jMax : LREAL;  
END_VAR
THIS^.p0 := p0;
THIS^.v0 := v0;
THIS^.a0 := a0;
THIS^.tf := tf;
THIS^.pf := pf;
THIS^.vf := vf;
THIS^.af := af;
THIS^._vMax := vMax;
THIS^._vMin := vMin;
THIS^._aMax := aMax;
THIS^._aMin := aMin;
THIS^._jMax := jMax;

pd := pf - p0;
tf_tf := tf * tf;
tf_p3 := tf_tf * tf;
tf_p4 := tf_tf * tf_tf;

vd := vf - v0;
vd_vd := vd * vd;
v0_v0 := v0 * v0;
vf_vf := vf * vf;

ad := af - a0;
ad_ad := ad * ad;
a0_a0 := a0 * a0;
af_af := af * af;

a0_p3 := a0 * a0_a0;
a0_p4 := a0_a0 * a0_a0;
a0_p5 := a0_p3 * a0_a0;
a0_p6 := a0_p4 * a0_a0;
af_p3 := af * af_af;
af_p4 := af_af * af_af;
af_p5 := af_p3 * af_af;
af_p6 := af_p4 * af_af;

// max values needs to be invariant to plus minus sign change
jMax_jMax := jMax * jMax;

g1 := -pd + tf*v0;
g2 := -2*pd + tf*(v0 + vf);
END_METHOD

METHOD PRIVATE time_acc0 : BOOL
VAR_IN_OUT
  Profile : ProfileDesc;
END_VAR
VAR_INPUT
  vMax, vMin, aMax, aMin, jMax : LREAL;
END_VAR
VAR
  h0a, h0b, h0c, h1, h2 : LREAL;
END_VAR
h1 := SQRT(ad_ad/(2*jMax_jMax) - ad*(aMax - a0)/(jMax_jMax) + (aMax*tf - vd)/jMax);

Profile.t[0] := (aMax - a0)/jMax;
Profile.t[1] := tf - ad/jMax - 2*h1;
Profile.t[2] := h1;
Profile.t[3] := 0;
Profile.t[4] := (af - aMax)/jMax + h1;
Profile.t[5] := 0;
Profile.t[6] := 0;

time_acc0 := profile.CheckWithTiming(ProfileJerkSigns.Udud, ProfileLimits.None, tf, jMax, vMax, vMin, aMax, aMin);
IF time_acc0
THEN
  RETURN;
END_IF        


// a3 != 0
// UDDU Solution 1
h0a := a0_p3 + 2*af_p3 - 6*(af_af + aMax*aMax)*aMax - 6*(a0 + af)*aMax*jMax*tf + 9*aMax*aMax*(af + jMax*tf) + 3*a0*aMax*(-2*af + 3*aMax) + 3*a0_a0*(af - 2*aMax + jMax*tf) - 6*jMax_jMax*g1 + 6*(af - aMax)*jMax*vd - 3*aMax*jMax_jMax*tf_tf;
h0b := a0_a0 + af_af + 2*(aMax*aMax - (a0 + af)*aMax + jMax*(vd - aMax*tf));
h1 := 4*h0a*h0a - 18*h0b*h0b*h0b;
IF h1 >= 0
THEN
  h1 := ABS(jMax)/jMax*SQRT(h1);
  h2 := 6*jMax*h0b;
  
  Profile.t[0] := (-a0 + aMax)/jMax;
  Profile.t[1] := ad/jMax - 2 * Profile.t[0] - (2*h0a - h1)/h2 + tf;
  Profile.t[2] := -(2*h0a + h1)/h2;
  Profile.t[3] := (2*h0a - h1)/h2;
  Profile.t[4] := tf - (Profile.t[0] + Profile.t[1] + Profile.t[2] + Profile.t[3]);
  Profile.t[5] := 0;
  Profile.t[6] := 0;
  
  time_acc0 := Profile.CheckWithTiming(ProfileJerkSigns.Uddu, ProfileLimits.ACC0, tf, jMax, vMax, vMin, aMax, aMin);
END_IF
END_METHOD

METHOD PRIVATE time_acc0_acc1 : BOOL
VAR_IN_OUT
  Profile : ProfileDesc;
END_VAR
VAR_INPUT
  vMax, vMin, aMax, aMin, jMax : LREAL;
END_VAR
VAR
  h0a : LREAL;
  h1, h2, h3, jf : LREAL;
END_VAR
IF (ABS(a0) < Constants.DoubleEpsilon AND_THEN ABS(af) < Constants.DoubleEpsilon)
THEN
  h1 := 2*aMin*(-pd + tf*v0) + vd_vd + aMax*(2*pd + aMin*tf_tf - 2*tf*vf);
  h2 := ((aMax - aMin)*(-aMin*vd + aMax*(aMin*tf - vd)));

  IF h1 <> 0
  THEN
    jf := h2/h1;
    Profile.t[0] := aMax/jf;
    Profile.t[1] := (-2*aMax*h1 + aMin*aMin*(-2*pd + tf*(v0 + vf)))/h2;
    Profile.t[2] := Profile.t[0];
    Profile.t[3] := 0;
    Profile.t[4] := -aMin/jf;
    Profile.t[5] := tf - (2*Profile.t[0] + Profile.t[1] + 2*Profile.t[4]);
    Profile.t[6] := Profile.t[4];

    time_acc0_acc1 := Profile.CheckWithTiming2(ProfileJerkSigns.Uddu, ProfileLimits.Acc0Acc1, tf, jf, vMax, vMin, aMax, aMin, jMax);
    RETURN;
  END_IF
END_IF

h1 := 144*Power2((aMax - aMin)*(-aMin*vd + aMax*(aMin*tf - vd)) - af_af*(aMax*tf - vd) + 2*af*aMin*(aMax*tf - vd) + a0_a0*(aMin*tf + v0 - vf) - 2*a0*aMax*(aMin*tf - vd)) + 48*ad*(3*a0_p3 - 3*af_p3 + 12*aMax*aMin*(-aMax + aMin) + 4*af_af*(aMax + 2*aMin) + a0*(-3*af_af - 8*af*aMax + 6*aMax*aMax + 8*af*aMin + 12*aMax*aMin - 6*aMin*aMin) + 6*af*(aMax*aMax - 2*aMax*aMin - aMin*aMin) + a0_a0*(3*af - 4*(2*aMax + aMin)))*(2*aMin*(-pd + tf*v0) + vd*vd + aMax*(2*pd + aMin*tf*tf - 2*tf*vf));
IF h1 >= 0
THEN
  h1 := SQRT(h1);
  jf := -(3*af_af*aMax*tf - 3*a0_a0*aMin*tf - 6*ad*aMax*aMin*tf + 3*aMax*aMin*(aMin - aMax)*tf + 3*(a0_a0 - af_af)*vd + 6*af*aMin*vd - 6*a0*aMax*vd + 3*(aMax*aMax - aMin*aMin)*vd + h1/4)/(6*(2*aMin*(-pd + tf*v0) + vd*vd + aMax*(2*pd + aMin*tf_tf - 2*tf*vf)));
  
  IF ABS(jf) > Constants.Epsilon
  THEN
  
    Profile.t[0] := (aMax - a0)/jf;
    Profile.t[1] := (a0_a0 - af_af + 2*ad*aMin - 2*(aMax*aMax - 2*aMax*aMin + aMin*aMin + aMin*jf*tf - jf*vd))/(2*(aMax - aMin)*jf);
    Profile.t[2] := aMax/jf;
    Profile.t[3] := 0;
    Profile.t[4] := -aMin/jf;
    Profile.t[5] := tf - (Profile.t[0] + Profile.t[1] + Profile.t[2] + 2*Profile.t[4] + af/jf);
    Profile.t[6] := Profile.t[4] + af/jf;
    
    time_acc0_acc1 := Profile.CheckWithTiming2(ProfileJerkSigns.Uddu, ProfileLimits.Acc0Acc1, tf, jf, vMax, vMin, aMax, aMin, jMax);
    IF time_acc0_acc1
    THEN
      RETURN;
    END_IF
  
	END_IF  
END_IF


// Profile UDDU, Solution 1
{}
  profile.t[0] := (-a0 + aMax)/jMax;
  profile.t[1] := -((af_af - a0_a0)/2 + aMax*aMax + aMin*aMin - ad*aMin - 2*aMax*aMin + jMax*(aMin*tf - vd))/((aMax - aMin)*jMax);
  profile.t[2] := aMax/jMax;
  profile.t[3] := 0;
  profile.t[4] := -aMin/jMax;
  profile.t[5] := tf - (profile.t[0] + profile.t[1] + profile.t[2] + profile.t[3] + 2*profile.t[4] + af/jMax);
  profile.t[6] := profile.t[4] + af/jMax;
  
  time_acc0_acc1 := Profile.CheckWithTiming(ProfileJerkSigns.Uddu, ProfileLimits.Acc0Acc1, tf, jMax, vMax, vMin, aMax, aMin);
  IF time_acc0_acc1
  THEN
    RETURN;
  END_IF
{}
END_METHOD

METHOD PRIVATE time_acc0_acc1_vel : BOOL
VAR_IN_OUT
  Profile : ProfileDesc;
END_VAR
VAR_INPUT
  vMax, vMin, aMax, aMin, jMax : LREAL;
END_VAR
VAR_INST
  h0, h1, h2, h3 : LREAL;
END_VAR
// Profile UDDU, Solution 1
IF ((2*(aMax - aMin) + ad)/jMax < tf) THEN
  h1 := (a0_p4 + af_p4 - 4*a0_p3*(2*aMax + aMin)/3 - 4*af_p3*(aMax + 2*aMin)/3 + 2*(a0_a0 - af_af)*aMax*aMax + (4*a0*aMax - 2*a0_a0)*(af_af - 2*af*aMin + (aMin - aMax)*aMin + 2*jMax*(aMin*tf - vd)) + 2*af_af*(aMin*aMin + 2*jMax*(aMax*tf - vd)) + 4*jMax*(2*aMin*(af*vd + jMax*g1) + (aMax*aMax - aMin*aMin)*vd + jMax*vd_vd) + 8*aMax*jMax_jMax*(pd - tf*vf))/(aMax*aMin) + 4*af_af + 2*a0_a0 + (4*af + aMax - aMin)*(aMax - aMin) + 4*jMax*(aMin - aMax + jMax*tf - 2*af)*tf;
  IF h1 >= 0
  THEN
    h1 := SQRT(h1) * ABS(jMax)/jMax;
    
    Profile.t[0] := (-a0 + aMax)/jMax;
    Profile.t[1] := (-(af_af - a0_a0 + 2*aMax*aMax + aMin*(aMin - 2*ad - 3*aMax) + 2*jMax*(aMin*tf - vd)) + aMin*h1)/(2*(aMax - aMin)*jMax);
    Profile.t[2] := aMax/jMax;
    Profile.t[3] := (aMin - aMax + h1)/(2*jMax);
    Profile.t[4] := -aMin/jMax;
    Profile.t[5] := tf - (Profile.t[0] + Profile.t[1] + Profile.t[2] + Profile.t[3] + 2*Profile.t[4] + af/jMax);
    Profile.t[6] := Profile.t[4] + af/jMax;
    
    time_acc0_acc1_vel := Profile.CheckWithTiming(ProfileJerkSigns.Uddu, ProfileLimits.Acc0Acc1Vel, tf, jMax, vMax, vMin, aMax, aMin);
    IF time_acc0_acc1_vel
    THEN
      RETURN;
    END_IF
  END_IF
END_IF

// Profile UDUD
Profile.t[1] := (3*(a0_p4 + af_p4) - 4*(a0_p3 + af_p3)*aMax - 4*af_p3*aMax + 24*(a0 + af)*aMax*aMax*aMax - 6*(af_af + a0_a0)*(aMax*aMax - 2*jMax*vd) + 6*a0_a0*(af_af - 2*af*aMax - 2*aMax*jMax*tf) - 12*aMax*aMax*(2*aMax*aMax - 2*aMax*jMax*tf + jMax*vd) - 24*af*aMax*jMax*vd + 12*jMax_jMax*(2*aMax*g1 + vd_vd))/(12*aMax*jMax*(a0_a0 + af_af - 2*(a0 + af)*aMax + 2*(aMax*aMax - aMax*jMax*tf + jMax*vd)));
Profile.t[2] := aMax/jMax;
Profile.t[3] := (-a0_a0 - af_af + 2*aMax*(a0 + af - 2*aMax) - 2*jMax*vd)/(2*aMax*jMax) + tf;
Profile.t[4] := Profile.t[2];
Profile.t[5] := tf - (Profile.t[0] + Profile.t[1] + Profile.t[2] + Profile.t[3] + 2*Profile.t[4] - af/jMax);
Profile.t[6] := Profile.t[4] - af/jMax;

time_acc0_acc1_vel := Profile.CheckWithTiming(ProfileJerkSigns.Udud, ProfileLimits.Acc0Acc1Vel, tf, jMax, vMax, vMin, aMax, aMin);
END_METHOD

METHOD PRIVATE time_acc0_vel : BOOL
VAR_IN_OUT
  Profile : ProfileDesc;
END_VAR
VAR_INPUT
  vMax, vMin, aMax, aMin, jMax : LREAL;
END_VAR
VAR
  ph1, ph2, ph3, ph4 : LREAL;
  polynom : ARRAY[0..4] OF LREAL;
  t : LREAL; 
  orig, deriv : LREAL;
  h1 : LREAL;
  i : INT;  
END_VAR
IF (tf < MAX((-a0 + aMax)/jMax, 0.0) + MAX(aMax/jMax, 0.0))
THEN
  RETURN;
END_IF

ph1 := 12*jMax*(-aMax*aMax*vd - jMax*vd_vd + 2*aMax*jMax*(-pd + tf*vf));

polynom[1] := (2*aMax)/jMax;
polynom[2] := (a0_a0 - af_af + 2*ad*aMax + aMax*aMax + 2*jMax*(vd - aMax*tf))/jMax_jMax;
polynom[3] := 0;
polynom[4] := -(-3*(a0_p4 + af_p4) + 4*(af_p3 + 2*a0_p3)*aMax - 12*a0*aMax*(af_af - 2*jMax*vd) + 6*a0_a0*(af_af - aMax*aMax - 2*jMax*vd) + 6*af_af*(aMax*aMax - 2*aMax*jMax*tf + 2*jMax*vd) + ph1)/(12*jMax_jMax*jMax_jMax);

t_min := -af/jMax;
t_max := MIN(tf - aMax/jMax, -aMin/jMax);
        
Roots.SolveQuartMonic(ADR(polynom[1]), 4, rootCount:=d_extremasCount, roots:=d_extremas);
FOR i:=0 TO d_extremasCount
DO
  t := d_extremas[i];
  IF t < t_min OR_ELSE t > t_max
  THEN
    CONTINUE;
  END_IF

  // Single Newton step (regarding pd)
  IF (t > Constants.DoubleEpsilon)
  THEN
    h1 := jMax*t*t + vd;
    orig := (-3*(a0_p4 + af_p4) + 4*(af_p3 + 2*a0_p3)*aMax - 24*af*aMax*jMax_jMax*t*t - 12*a0*aMax*(af_af - 2*jMax*h1) + 6*a0_a0*(af_af - aMax*aMax - 2*jMax*h1) + 6*af_af*(aMax*aMax - 2*aMax*jMax*tf + 2*jMax*h1) - 12*jMax*(aMax*aMax*h1 + jMax*h1*h1 + 2*aMax*jMax*(pd + jMax*t*t*(t - tf) - tf*vf)))/(24*aMax*jMax_jMax);                
    deriv := -t*(a0_a0 - af_af + 2*aMax*(ad - jMax*tf) + aMax*aMax + 3*aMax*jMax*t + 2*jMax*h1)/aMax;
  
    IF ABS(deriv) < Constants.DoubleEpsilon
    THEN
      CONTINUE;
    END_IF  

    t := t - orig / deriv;	  
  END_IF


  h1 := ((a0_a0 - af_af)*0.5 + jMax*(jMax*t*t + vd))/aMax;

  Profile.t[0] := (-a0 + aMax)/jMax;
  Profile.t[1] := (h1 - aMax)/jMax;
  Profile.t[2] := aMax/jMax;
  Profile.t[3] := tf - (h1 + ad + aMax)/jMax - 2*t;
  Profile.t[4] := t;
  Profile.t[5] := 0;
  Profile.t[6] := af/jMax + t;

  time_acc0_vel := Profile.CheckWithTiming(ProfileJerkSigns.Uddu, ProfileLimits.Acc0Vel, tf, jMax, vMax, vMin, aMax, aMin);
  IF time_acc0_vel
  THEN
    RETURN;
  END_IF
END_FOR
        

polynom[1] := (-2*aMax)/jMax;
polynom[2] := -(a0_a0 + af_af - 2*(a0 + af)*aMax + aMax*aMax + 2*jMax*(vd - aMax*tf))/jMax_jMax;
polynom[3] := 0;
polynom[4] := (3*(a0_p4 + af_p4) - 4*(af_p3 + 2*a0_p3)*aMax + 6*a0_a0*(af_af + aMax*aMax + 2*jMax*vd) - 12*a0*aMax*(af_af + 2*jMax*vd) + 6*af_af*(aMax*aMax - 2*aMax*jMax*tf + 2*jMax*vd) - ph1)/(12*jMax_jMax*jMax_jMax);

t_min := af/jMax;
t_max := MIN(tf - (2*aMax - a0)/jMax, -aMin/jMax);
        
Roots.SolveQuartMonic(ADR(polynom[1]), 4, rootCount:=d_extremasCount, roots:=d_extremas);
FOR i:=0 TO d_extremasCount
DO
  t := d_extremas[i];
  IF t < t_min OR_ELSE t > t_max
  THEN
    CONTINUE;
  END_IF

  // Single Newton step (regarding pd)
  h1 := jMax*t*t - vd;
  orig := -(3*(a0_p4 + af_p4) - 4*(2*a0_p3 + af_p3)*aMax + 24*af*aMax*jMax_jMax*t*t - 12*a0*aMax*(af_af - 2*jMax*h1) + 6*a0_a0*(af_af + aMax*aMax - 2*jMax*h1) + 6*af_af*(aMax*aMax - 2*jMax*(tf*aMax + h1)) + 12*jMax*(-aMax*aMax*h1 + jMax*h1*h1 - 2*aMax*jMax*(-pd + jMax*t*t*(t - tf) + tf*vf)))/(24*aMax*jMax_jMax);
  deriv := t*(a0_a0 + af_af - 2*jMax*h1 - 2*(a0 + af + jMax*tf)*aMax + aMax*aMax + 3*aMax*jMax*t)/aMax;
  
  IF ABS(deriv) < Constants.DoubleEpsilon
  THEN
    CONTINUE;
  END_IF    
  
  t := t - orig / deriv;
  
  h1 := ((a0_a0 + af_af)*0.5 + jMax*(vd - jMax*t*t))/aMax;
  Profile.t[0] := (-a0 + aMax)/jMax;
  Profile.t[1] := (h1 - aMax)/jMax;
  Profile.t[2] := aMax/jMax;
  Profile.t[3] := tf - (h1 - a0 - af + aMax)/jMax - 2*t;
  Profile.t[4] := t;
  Profile.t[5] := 0;
  Profile.t[6] := -(af/jMax) + t;

  time_acc0_vel := Profile.CheckWithTiming(ProfileJerkSigns.Udud, ProfileLimits.Acc0Vel, tf, jMax, vMax, vMin, aMax, aMin);
  IF time_acc0_vel
  THEN
    RETURN;
  END_IF
END_FOR
END_METHOD

METHOD PRIVATE time_acc1 : BOOL
VAR_IN_OUT
  Profile : ProfileDesc;
END_VAR
VAR_INPUT
  vMax, vMin, aMax, aMin, jMax : LREAL;
END_VAR
VAR
  h0, h0a, h0b, h0c, h1, h2 : LREAL;
END_VAR
// a3 != 0
// Case UDDU
h0 := jMax_jMax*(a0_p4 + af_p4 - 4*af_p3*jMax*tf + 6*af_af*jMax_jMax*tf_tf - 4*a0_p3*(af - jMax*tf) + 6*a0_a0*(af - jMax*tf)*(af - jMax*tf) + 24*af*jMax_jMax*(-pd + tf*v0) - 4*a0*(af_p3 - 3*af_af*jMax*tf + 6*jMax_jMax*(-pd + tf*vf)) - 12*jMax_jMax*(-vd_vd + jMax*tf*(-2*pd + tf*(v0 + vf))))/3;
h1 := (a0_a0 + af_af - 2*a0*af - 2*ad*jMax*tf + 2*h0)/jMax_jMax + tf_tf;

IF h0 >= 0 AND_THEN h1 >= 0
THEN
  h0 := SQRT(h0)/jMax;
  h1 := SQRT(h1);
  
  Profile.t[0] := -(a0_a0 + af_af + 2*a0*(jMax*tf - af) - 2*jMax*vd + h0)/(2*jMax*(-ad + jMax*tf));
  Profile.t[1] := 0;
  Profile.t[2] := (tf - h1)/2 - ad/(2*jMax);
  Profile.t[3] := 0;
  Profile.t[4] := 0;
  Profile.t[5] := h1;
  Profile.t[6] := tf - (profile.t[0] + profile.t[2] + profile.t[5]);
  
  time_acc1 := Profile.CheckWithTiming(ProfileJerkSigns.Uddu, ProfileLimits.Acc1, tf, jMax, vMax, vMin, aMax, aMin);
  IF time_acc1
  THEN
    RETURN;
  END_IF
END_IF

// Case UDUD
h0 := jMax_jMax*(a0_p4 + af_p4 + 4*(af_p3 - a0_p3)*jMax*tf + 6*af_af*jMax_jMax*tf_tf + 6*a0_a0*(af + jMax*tf)*(af + jMax*tf) + 24*af*jMax_jMax*(-pd + tf*v0) - 4*a0*(a0_a0*af + af_p3 + 3*af_af*jMax*tf + 6*jMax_jMax*(-pd + tf*vf)) + 12*jMax_jMax*(vd_vd + jMax*tf*(-2*pd + tf*(v0 + vf))))/3;
h1 := (a0_a0 + af_af - 2*a0*af + 2*ad*jMax*tf + 2*h0)/jMax_jMax + tf_tf;

IF h0 >= 0 AND_THEN h1 >= 0
THEN
  h0 := SQRT(h0)/jMax;
  h1 := SQRT(h1);
  
  Profile.t[0] := 0;
  Profile.t[1] := 0;
  Profile.t[2] := -(a0_a0 + af_af - 2*a0*af + 2*jMax*(vd - a0*tf) + h0)/(2*jMax*(ad + jMax*tf));
  Profile.t[3] := 0;
  Profile.t[4] := ad/(2*jMax) + (tf - h1)/2;
  Profile.t[5] := h1;
  Profile.t[6] := tf - (profile.t[5] + profile.t[4] + profile.t[2]);
  
  time_acc1 := profile.CheckWithTiming(ProfileJerkSigns.Udud, ProfileLimits.Acc1, tf, jMax, vMax, vMin, aMax, aMin);
  IF time_acc1
  THEN
    RETURN;
  END_IF
END_IF

// Case UDDU, Solution 2
h0a := a0_p3 - af_p3 - 3*a0_a0*aMin + 3*aMin*aMin*(a0 + jMax*tf) + 3*af*aMin*(-aMin - 2*jMax*tf) - 3*af_af*(-aMin - jMax*tf) - 3*jMax_jMax*(-2*pd - aMin*tf_tf + 2*tf*vf);
h0b := a0_a0 + af_af - 2*(a0 + af)*aMin + 2*(aMin*aMin - jMax*(-aMin*tf + vd));
h0c := a0_p4 + 3*af_p4 - 4*(a0_p3 + 2*af_p3)*aMin + 6*a0_a0*aMin*aMin + 6*af_af*(aMin*aMin - 2*jMax*vd) + 12*jMax*(2*aMin*jMax*g1 - aMin*aMin*vd + jMax*vd_vd) + 24*af*aMin*jMax*vd - 4*a0*(af_p3 - 3*af*aMin*(-aMin - 2*jMax*tf) + 3*af_af*(-aMin - jMax*tf) + 3*jMax*(-aMin*aMin*tf + jMax*(-2*pd - aMin*tf_tf + 2*tf*vf)));
h1 := 4*h0a*h0a - 6*h0b*h0c;
IF h1 >= 0
THEN
  h1 := ABS(jMax)/jMax*SQRT(h1);
  h2 := 6*jMax*h0b;
	
  Profile.t[0] := 0;
  Profile.t[1] := 0;
  Profile.t[2] := (2*h0a + h1)/h2;
  Profile.t[3] := -(a0_a0 + af_af - 2*(a0 + af)*aMin + 2*(aMin*aMin + aMin*jMax*tf - jMax*vd))/(2*jMax*(a0 - aMin - jMax*Profile.t[2]));
  Profile.t[4] := (a0 - aMin)/jMax - Profile.t[2];
  Profile.t[5] := tf - (Profile.t[2] + Profile.t[3] + Profile.t[4] + (af - aMin)/jMax);
  Profile.t[6] := (af - aMin)/jMax;
	
  time_acc1 := Profile.CheckWithTiming(ProfileJerkSigns.Uddu, ProfileLimits.Acc1, tf, jMax, vMax, vMin, aMax, aMin);
  IF (time_acc1)
  THEN
    RETURN;
  END_IF
END_IF
    
// Case UDUD, Solution 1
h0a := -a0_p3 + af_p3 + 3*(a0_a0 - af_af)*aMax - 3*ad*aMax*aMax - 6*af*aMax*jMax*tf + 3*af_af*jMax*tf + 3*jMax*(aMax*aMax*tf + jMax*(-2*pd - aMax*tf_tf + 2*tf*vf));
h0b := a0_a0 - af_af + 2*ad*aMax + 2*jMax*(aMax*tf - vd);
h0c := a0_p4 + 3*af_p4 - 4*(a0_p3 + 2*af_p3)*aMax + 6*a0_a0*aMax*aMax - 24*af*aMax*jMax*vd + 12*jMax*(2*aMax*jMax*g1 + jMax*vd_vd + aMax*aMax*vd) + 6*af_af*(aMax*aMax + 2*jMax*vd) - 4*a0*(af_p3 + 3*af*aMax*(aMax - 2*jMax*tf) - 3*af_af*(aMax - jMax*tf) + 3*jMax*(aMax*aMax*tf + jMax*(-2*pd - aMax*tf_tf + 2*tf*vf)));
h1 := 4*h0a*h0a - 6*h0b*h0c;
IF h1 >= 0
THEN
	h1 := ABS(jMax)/jMax*SQRT(h1);
	h2 := 6*jMax*h0b;
	
	Profile.t[0] := 0;
	Profile.t[1] := 0;
	Profile.t[2] := -(2*h0a + h1)/h2;
	Profile.t[3] := 2*h1/h2;
	Profile.t[4] := (aMax - a0)/jMax + Profile.t[2];
	Profile.t[5] := tf - (Profile.t[2] + Profile.t[3] + Profile.t[4] + (-af + aMax)/jMax);
	Profile.t[6] := (-af + aMax)/jMax;
	
	time_acc1 := Profile.CheckWithTiming(ProfileJerkSigns.Udud, ProfileLimits.Acc1, tf, jMax, vMax, vMin, aMax, aMin);
	IF (time_acc1)
	THEN
	  RETURN;
	END_IF
END_IF
END_METHOD

METHOD PRIVATE time_acc1_vel : BOOL
VAR_IN_OUT
  Profile : ProfileDesc;
END_VAR
VAR_INPUT
  vMax, vMin, aMax, aMin, jMax : LREAL;
END_VAR
VAR
  h0, ph1, ph2, ph3, ph4 : LREAL;
  polynom : ARRAY[0..4] OF LREAL; 
  t : LREAL; 
  orig, deriv : LREAL;
  h1 : LREAL;
  i : INT;
END_VAR
// Profile UDDU
ph1 := a0_a0 + af_af - aMin*(a0 + 2*af - aMin) - 2*jMax*(vd - aMin*tf);
ph2 := 2*aMin*(jMax*g1 + af*vd) - aMin*aMin*vd + jMax*vd_vd;
ph3 := af_af + aMin*(aMin - 2*af) - 2*jMax*(vd - aMin*tf);

polynom[1] := (2*(2*a0 - aMin))/jMax;
polynom[2] := (4*a0_a0 + ph1 - 3*a0*aMin)/jMax_jMax;
polynom[3] := (2*a0*ph1)/(jMax_jMax*jMax);
polynom[4] := (3*(a0_p4 + af_p4) - 4*(a0_p3 + 2*af_p3)*aMin + 6*af_af*(aMin*aMin - 2*jMax*vd) + 12*jMax*ph2 + 6*a0_a0*ph3)/(12*jMax_jMax*jMax_jMax);

t_min := -a0/jMax;
t_max := MIN((tf + 2*aMin/jMax - (a0 + af)/jMax)/2, (aMax - a0)/jMax);

Roots.SolveQuartMonic(ADR(polynom[1]), 4, rootCount:=d_extremasCount, roots:=d_extremas);
FOR i:=0 TO d_extremasCount
DO
  t := d_extremas[i];
  IF t < t_min OR_ELSE t > t_max
  THEN
    CONTINUE;
  END_IF

  // Single Newton step (regarding pd)
  IF ABS(a0 + jMax*t) > 16 * Constants.DoubleEpsilon
  THEN
    h0 := jMax*t*t;
    orig := -pd + (3*(a0_p4 + af_p4) - 8*af_p3*aMin - 4*a0_p3*aMin + 6*af_af*(aMin*aMin + 2*jMax*(h0 - vd)) + 6*a0_a0*(af_af - 2*af*aMin + aMin*aMin + 2*aMin*jMax*(-2*t + tf) + 2*jMax*(5*h0 - vd)) + 24*a0*jMax*t*(a0_a0 + af_af - 2*af*aMin + aMin*aMin + 2*jMax*(aMin*(-t + tf) + h0 - vd)) - 24*af*aMin*jMax*(h0 - vd) + 12*jMax*(aMin*aMin*(h0 - vd) + jMax*(h0 - vd)*(h0 - vd)))/(24*aMin*jMax_jMax) + h0*(tf - t) + tf*v0;
    deriv := (a0 + jMax*t)*((a0_a0 + af_af)/(aMin*jMax) + (aMin - a0 - 2*af)/jMax + (4*a0*t + 2*h0 - 2*vd)/aMin + 2*tf - 3*t);
                
    IF ABS(deriv) < Constants.DoubleEpsilon
    THEN
      CONTINUE;
    END_IF    
  
    t := t - orig / deriv;
  END_IF
  
  h1 := -((a0_a0 + af_af)*0.5 + jMax*(-vd + 2*a0*t + jMax*t*t))/aMin;

  Profile.t[0] := t;
  Profile.t[1] := 0;
  Profile.t[2] := a0/jMax + t;
  Profile.t[3] := tf - (h1 - aMin + a0 + af)/jMax - 2*t;
  Profile.t[4] := -aMin/jMax;
  Profile.t[5] := (h1 + aMin)/jMax;
  Profile.t[6] := Profile.t[4] + af/jMax;

  time_acc1_vel := Profile.CheckWithTiming(ProfileJerkSigns.Uddu, ProfileLimits.Acc1Vel, tf, jMax, vMax, vMin, aMax, aMin);
  IF time_acc1_vel
  THEN
    RETURN;
	END_IF
END_FOR



// Profile UDUD
ph1 := a0_a0 - af_af + (2*af - a0)*aMax - aMax*aMax - 2*jMax*(vd - aMax*tf);
ph2 := aMax*aMax + 2*jMax*vd;
ph3 := af_af + ph2 - 2*aMax*(af + jMax*tf);
ph4 := 2*aMax*jMax*g1 + aMax*aMax*vd + jMax*vd_vd;

polynom[1] := (4*a0 - 2*aMax)/jMax;
polynom[2] := (4*a0_a0 - 3*a0*aMax + ph1)/jMax_jMax;
polynom[3] := (2*a0*ph1)/(jMax_jMax*jMax);
polynom[4] := (3*(a0_p4 + af_p4) - 4*(a0_p3 + 2*af_p3)*aMax - 24*af*aMax*jMax*vd + 12*jMax*ph4 - 6*a0_a0*ph3 + 6*af_af*ph2)/(12*jMax_jMax*jMax_jMax);

t_min := -a0/jMax;
t_max := MIN((tf + ad/jMax - 2*aMax/jMax)/2, (aMax - a0)/jMax);
        
Roots.SolveQuartMonic(ADR(polynom[1]), 4, rootCount:=d_extremasCount, roots:=d_extremas);
FOR i:=0 TO d_extremasCount
DO
  t := d_extremas[i];
  IF t > t_max OR_ELSE t < t_min
  THEN
    CONTINUE;
	END_IF

  h1 := ((a0_a0 - af_af)*0.5 + jMax_jMax*t*t - jMax*(vd - 2*a0*t))/aMax;

  Profile.t[0] := t;
  Profile.t[1] := 0;
  Profile.t[2] := t + a0/jMax;
  Profile.t[3] := tf + (h1 + ad - aMax)/jMax - 2*t;
  Profile.t[4] := aMax/jMax;
  Profile.t[5] := -(h1 + aMax)/jMax;
  Profile.t[6] := Profile.t[4] - af/jMax;

  time_acc1_vel := Profile.CheckWithTiming(ProfileJerkSigns.Udud, ProfileLimits.Acc1Vel, tf, jMax, vMax, vMin, aMax, aMin);
  IF time_acc1_vel
  THEN
    RETURN;
	END_IF
END_FOR
END_METHOD

METHOD PRIVATE time_none : BOOL
VAR_IN_OUT
  Profile : ProfileDesc;
END_VAR
VAR_INPUT
  vMax, vMin, aMax, aMin, jMax : LREAL;
END_VAR
VAR
  t, h0, h1, h2, h3, orig, deriv, jf: LREAL;
  polynom : ARRAY[0..4] OF LREAL;
  i : INT;
  ph0, ph1, ph2, ph3, ph4, ph5, ph6, ph7 : LREAL;
END_VAR
IF (ABS(v0) < Constants.DoubleEpsilon AND_THEN ABS(a0) < Constants.DoubleEpsilon AND_THEN ABS(af) < Constants.DoubleEpsilon)
THEN
  h1 := SQRT(tf_tf*vf_vf + (4*pd - tf*vf)*(4*pd - tf*vf));
  jf := 4*(4*pd - 2*tf*vf + h1)/tf_p3;
  
  Profile.t[0] := tf/4;
  Profile.t[1] := 0;
  Profile.t[2] := 2*Profile.t[0];
  Profile.t[3] := 0;
  Profile.t[4] := 0;
  Profile.t[5] := 0;
  Profile.t[6] := Profile.t[0];
  time_none := Profile.CheckWithTiming2(ProfileJerkSigns.Uddu, ProfileLimits.None, tf, jf, vMax, vMin, aMax, aMin, jMax);
  IF time_none THEN
    RETURN;
  END_IF
END_IF

h1 := 16*pd*(pd - tf*(v0 + vf)) + tf_tf*(5*v0_v0 + 6*v0*vf + 5*vf_vf);
IF (ABS(a0) < Constants.DoubleEpsilon AND_THEN ABS(af) < Constants.DoubleEpsilon) AND_THEN vd > Constants.DoubleEpsilon AND_THEN h1 >= 0
THEN
  h1 := SQRT(h1);
  jf := 4*(4*pd - 2*tf*(v0 + vf) - h1)/tf_p3;
  
  Profile.t[0] := (tf*(v0 + 3*vf) - 4*pd)/(4*vd);
  Profile.t[1] := 0;
  Profile.t[2] := tf*0.5;
  Profile.t[3] := 0;
  Profile.t[4] := 0;
  Profile.t[5] := 0;
  Profile.t[6] := Profile.t[4];

  time_none := Profile.CheckWithTiming2(ProfileJerkSigns.UDDU, ProfileLimits.None, tf, jf, vMax, vMin, aMax, aMin, jMax);
  IF time_none
  THEN
    RETURN;
  END_IF
END_IF


// Is that really needed?
// Profiles with a3 != 0, Solution UDDU

// First acc, then constant
polynom[1] := -2*tf;
polynom[2] := 2*vd/jMax + tf_tf;
polynom[3] := 4*(pd - tf*vf)/jMax;
polynom[4] := (vd_vd + jMax*tf*g2)/(jMax_jMax);
Roots.SolveQuartMonic(ADR(polynom[1]), 4, rootCount:=d_extremasCount, roots:=d_extremas);
FOR i:=0 TO d_extremasCount
DO
  t := d_extremas[i];
  IF t > tf * 0.5 OR_ELSE t > (aMax - a0)/jMax
  THEN
    CONTINUE;
  END_IF

  // Single Newton step (regarding pd)
  h1 := (jMax*t*(t - tf) + vd)/(jMax*(2*t - tf));
  h2 := (2*jMax*t*(t - tf) + jMax*tf_tf - 2*vd)/(jMax*(2*t - tf)*(2*t - tf));
  orig := (-2*pd + 2*tf*v0 + h1*h1*jMax*(tf - 2*t) + jMax*tf*(2*h1*t - t*t - (h1 - t)*tf))*0.5;
  deriv := (jMax*tf*(2*t - tf)*(h2 - 1))*0.5 + h1*jMax*(tf - (2*t - tf)*h2 - h1);
  
  IF ABS(deriv) < Constants.DoubleEpsilon
  THEN
    CONTINUE;
  END_IF    
  
  t := t - orig / deriv;
  
  Profile.t[0] := t;
  Profile.t[1] := 0;
  Profile.t[2] := (jMax*t*(t - tf) + vd)/(jMax*(2*t - tf));
  Profile.t[3] := tf - 2*t;
  Profile.t[4] := t - Profile.t[2];
  Profile.t[5] := 0;
  Profile.t[6] := 0;
  
  time_none := Profile.CheckWithTiming2(ProfileJerkSigns.Uddu, ProfileLimits.None, tf, jMax, vMax, vMin, aMax, aMin, jMax);
  IF time_none
  THEN
    RETURN;
	END_IF
END_FOR


// First constant, then acc
ph1 := -jMax*(jMax*tf_tf + 4*vd);

polynom[1] := 2*jMax*(-4*pd + tf*(jMax*tf_tf - 2*v0 + 6*vf))/ph1;
polynom[2] := -(jMax_jMax*tf_p4 - 8*vd_vd + 4*jMax*tf*(-3*pd + tf*v0 + 2*tf*vf))/ph1;
polynom[3] := 4*(jMax*tf_tf*g1 - vd*(-2*pd - tf*v0 + 3*tf*vf))/ph1;
polynom[4] := -4*(jMax*g1*g1 + vd_vd*vd)/(jMax*ph1);

Roots.SolveQuartMonic(ADR(polynom[1]), 4, rootCount:=d_extremasCount, roots:=d_extremas);
FOR i:=0 TO d_extremasCount
DO
  t := d_extremas[i];
  IF t > tf OR_ELSE t > (aMax - a0)/jMax
  THEN
    CONTINUE;
  END_IF


  // Single Newton step (regarding pd)
  h1 := (jMax*t*(t - tf) - vd)/jMax;
  IF h1 <= 0
  THEN
  	CONTINUE;
  END_IF
  
  h1 := SQRT(h1);
  orig := (-2*pd + jMax*t*(t - tf)*tf + 2*tf*v0)*0.5 - (h1*h1*h1)/jMax - t*(jMax*t*(t - tf) - vd);
  deriv := (jMax*(-2*t + tf)*(6*h1 - 2*tf) - 4*jMax*t*(3*t - 2*tf))/4 + vd;
  
  IF ABS(deriv) < Constants.DoubleEpsilon
  THEN
    CONTINUE;
  END_IF    
  
  t := t - orig / deriv;
  
  h1 := (jMax*t*(t - tf) - vd)/jMax;
  IF h1 <= 0
  THEN
  	CONTINUE;
  END_IF
  
  h1 := SQRT(h1);
  
  // Solution 2 with aPlat
  Profile.t[0] := 0;
  Profile.t[1] := 0;
  Profile.t[2] := t;
  Profile.t[3] := tf - 2*t - 2*h1;
  Profile.t[4] := h1;
  Profile.t[5] := 0;
  Profile.t[6] := tf - (t + Profile.t[3] + Profile.t[4]);
  
  time_none := Profile.CheckWithTiming(ProfileJerkSigns.Uddu, ProfileLimits.None, tf, jMax, vMax, vMin, aMax, aMin);
  IF time_none 
  THEN
    RETURN; 
  END_IF
END_FOR

// UDUD T 0246
{}
  h0 := 2*jMax_jMax*(2*Power2(a0_p3 - af_p3 - 3*af_af*jMax*tf + 9*af*jMax_jMax*tf_tf - 3*a0_a0*(af + jMax*tf) + 3*a0*Power2(af + jMax*tf) + 3*jMax_jMax*(8*pd + jMax*tf_tf*tf - 8*tf*vf)) - 3*(a0_a0 + af_af - 2*af*jMax*tf - 2*a0*(af + jMax*tf) - jMax*(jMax*tf_tf + 4*v0 - 4*vf))*(a0_p4 + af_p4 + 4*af_p3*jMax*tf + 6*af_af*jMax_jMax*tf_tf - 3*jMax_jMax*jMax_jMax*tf_tf*tf_tf - 4*a0_p3*(af + jMax*tf) + 6*a0_a0*Power2(af + jMax*tf) - 12*af*jMax_jMax*(8*pd + jMax*tf_tf*tf - 8*tf*v0) + 48*jMax_jMax*vd_vd + 48*jMax_jMax*jMax*tf*(-2*pd + tf*(v0 + vf)) - 4*a0*(af_p3 + 3*af_af*jMax*tf - 9*af*jMax_jMax*tf_tf - 3*jMax_jMax*(8*pd + jMax*tf_tf*tf - 8*tf*vf))));
  IF h0 >= 0
  THEN
    h0 := SQRT(h0)/jMax;
    h1 := 12*jMax*(-a0_a0 - af_af + 2*af*jMax*tf + 2*a0*(af + jMax*tf) + jMax*(jMax*tf_tf + 4*v0 - 4*vf));
    h2 := -4*a0_p3 + 4*af_p3 + 12*a0_a0*af - 12*a0*af_af + 48*jMax_jMax*pd + 12*(a0_a0 - af_af)*jMax*tf - 24*jMax_jMax*tf*(v0 + vf) + 24*ad*jMax*vd;
    h3 := 2*a0_p3 - 2*af_p3 - 6*a0_a0*af + 6*a0*af_af;

    profile.t[0] := (h3 - 48*jMax_jMax*(tf*vf - pd) - 6*(a0_a0 + af_af)*jMax*tf + 12*a0*af*jMax*tf + 6*(a0 + 3*af + jMax*tf)*tf_tf*jMax_jMax - h0)/h1;
    profile.t[1] := 0;
    profile.t[2] := (h2 + h0)/h1;
    profile.t[3] := 0;
    profile.t[4] := (-h2 + h0)/h1;
    profile.t[5] := 0;
    profile.t[6] := (-h3 + 48*jMax_jMax*(tf*v0 - pd) - 6*(a0_a0 + af_af)*jMax*tf + 12*a0*af*jMax*tf + 6*(af + 3*a0 + jMax*tf)*tf_tf*jMax_jMax - h0)/h1;

    time_none := Profile.checkWithTiming(ProfileJerkSigns.Uddu, ProfileLimits.None, tf, jMax, vMax, vMin, aMax, aMin);
    IF time_none
    THEN
      RETURN;
    END_IF
  END_IF
{}

// Profiles with a3 != 0, Solution UDDU
// T 0234
ph1 := af + jMax*tf;
polynom[1] := -2*(ad + jMax*tf)/jMax;
polynom[2] := 2*(a0_a0 + af_af + jMax*(af*tf + vd) - 2*a0*ph1)/jMax_jMax + tf_tf;
polynom[3] := 2*(a0_p3 - af_p3 - 3*af_af*jMax*tf + 3*a0*ph1*(ph1 - a0) - 6*jMax_jMax*(-pd + tf*vf))/(3*jMax_jMax*jMax);
polynom[4] := (a0_p4 + af_p4 + 4*af_p3*jMax*tf - 4*a0_p3*ph1 + 6*a0_a0*ph1*ph1 + 24*jMax_jMax*af*g1 - 4*a0*(af_p3 + 3*af_af*jMax*tf + 6*jMax_jMax*(-pd + tf*vf)) + 6*jMax_jMax*af_af*tf_tf + 12*jMax_jMax*(vd_vd + jMax*tf*g2))/(12*jMax_jMax*jMax_jMax);
Roots.SolveQuartMonic(ADR(polynom[1]), 4, rootCount:=d_extremasCount, roots:=d_extremas);

t_min := ad/jMax;
t_max := MIN((aMax - a0)/jMax, (ad/jMax + tf) / 2);
            
FOR i:=0 TO d_extremasCount
DO
  t := d_extremas[i];
  IF t < t_min OR_ELSE t > t_max
  THEN
    CONTINUE;
	END_IF

  // Single Newton step (regarding pd)
  h0 := jMax*(2*t - tf) - ad;
  h1 := (ad_ad - 2*af*jMax*t + 2*a0*jMax*(t - tf) + 2*jMax*(jMax*t*(t - tf) + vd))/(2*jMax*h0);
  h2 := (-ad_ad + 2*jMax_jMax*(tf_tf + t*(t - tf)) + (a0 + af)*jMax*tf - ad*h0 - 2*jMax*vd)/(h0*h0);
  orig := (-a0_p3 + af_p3 + 3*ad_ad*jMax*(h1 - t) + 3*ad*jMax_jMax*(h1 - t)*(h1 - t) - 3*a0*af*ad + 3*jMax_jMax*(a0*tf_tf - 2*pd + 2*tf*v0 + h1*h1*jMax*(tf - 2*t) + jMax*tf*(2*h1*t - t*t - (h1 - t)*tf)))/(6*jMax_jMax);
  deriv := (h0*(-ad + jMax*tf)*(h2 - 1))/(2*jMax) + h1*(-ad + jMax*(tf - h1) - h0*h2);
  
  IF ABS(deriv) < Constants.DoubleEpsilon
  THEN
    CONTINUE;
	END_IF  
  
  t := t - orig / deriv;
  
  Profile.t[0] := t;
  Profile.t[1] := 0;
  Profile.t[2] := (ad_ad + 2*jMax*(-a0*tf - ad*t + jMax*t*(t - tf) + vd))/(2*jMax*(-ad + jMax*(2*t - tf)));
  Profile.t[3] := ad/jMax + tf - 2*t;
  Profile.t[4] := tf - (t + Profile.t[2] + Profile.t[3]);
  Profile.t[5] := 0;
  Profile.t[6] := 0;
  
  time_none := Profile.CheckWithTiming(ProfileJerkSigns.Uddu, ProfileLimits.None, tf, jMax, vMax, vMin, aMax, aMin);
  IF time_none
  THEN
    RETURN; 
  END_IF
END_FOR

// T 3456
{}
  h1 := 3*jMax*(ad_ad + 2*jMax*(a0*tf - vd));
  h2 := ad_ad + 2*jMax*(a0*tf - vd);
  h0 := 4*Power2(2*(a0_p3 - af_p3) - 6*a0_a0*(af - jMax*tf) + 6*jMax_jMax*(-pd + tf*v0) + 3*a0*(2*af_af - 2*jMax*af*tf + jMax_jMax*tf_tf) + 6*ad*jMax*vd) - 18*h2*h2*h2;
  IF h0 >= 0 AND_THEN h1 <> 0
  THEN
    h0 := SQRT(h0)/h1 * ABS(jMax)/jMax;
    
    profile.t[0] := 0;
    profile.t[1] := 0;
    profile.t[2] := 0;
    profile.t[3] := (af_p3 - a0_p3 + 3*(af_af - a0_a0)*jMax*tf - 3*ad*(a0*af + 2*jMax*vd) - 6*jMax_jMax*(-2*pd + tf*(v0 + vf)))/h1;
    profile.t[4] := (tf - profile.t[3] - h0)/2 - ad/(2*jMax);
    profile.t[5] := h0;
    profile.t[6] := (tf - profile.t[3] + ad/jMax - h0)/2;
    
    time_none := Profile.checkWithTiming(ProfileJerkSigns.Uddu, ProfileLimits.None, tf, jMax, vMax, vMin, aMax, aMin);
    IF time_none
    THEN
      RETURN;
    END_IF
	END_IF  
{}

// T 2346
ph1 := ad_ad + 2*(af + a0)*jMax*tf - jMax*(jMax*tf_tf + 4*vd);
ph2 := jMax*tf_tf*g1 - vd*(-2*pd - tf*v0 + 3*tf*vf);
ph3 := 5*af_af - 8*af*jMax*tf + 2*jMax*(2*jMax*tf_tf - vd);
ph4 := jMax_jMax*tf_p4 - 2*vd_vd + 8*jMax*tf*(-pd + tf*vf);
ph5 := (5*af_p4 - 8*af_p3*jMax*tf - 12*af_af*jMax*(jMax*tf_tf + vd) + 24*af*jMax_jMax*(-2*pd + jMax*tf_p3 + 2*tf*vf) - 6*jMax_jMax*ph4);
ph6 := -vd_vd + jMax*tf*(-2*pd + 3*tf*v0 - tf*vf) - af*g2;

polynom[1] := -(4*(a0_p3 - af_p3) - 12*a0_a0*(af - jMax*tf) + 6*a0*(2*af_af - 2*af*jMax*tf + jMax*(jMax*tf_tf - 2*vd)) + 6*af*jMax*(3*jMax*tf_tf + 2*vd) - 6*jMax_jMax*(-4*pd + jMax*tf_p3 - 2*tf*v0 + 6*tf*vf))/(3*jMax*ph1);
polynom[2] := -(-a0_p4 - af_p4 + 4*a0_p3*(af - jMax*tf) + a0_a0*(-6*af_af + 8*af*jMax*tf - 4*jMax*(jMax*tf_tf - vd)) + 2*af_af*jMax*(jMax*tf_tf + 2*vd) - 4*af*jMax_jMax*(-3*pd + jMax*tf_p3 + 2*tf*v0 + tf*vf) + jMax_jMax*(jMax_jMax*tf_p4 - 8*vd_vd + 4*jMax*tf*(-3*pd + tf*v0 + 2*tf*vf)) + 2*a0*(2*af_p3 - 2*af_af*jMax*tf + af*jMax*(-3*jMax*tf_tf - 4*vd) + jMax_jMax*(-6*pd + jMax*tf_p3 - 4*tf*v0 + 10*tf*vf)))/(jMax_jMax*ph1);
polynom[3] := -(a0_p5 - af_p5 + af_p4*jMax*tf - 5*a0_p4*(af - jMax*tf) + 2*a0_p3*ph3 + 4*af_p3*jMax*(jMax*tf_tf + vd) + 12*jMax_jMax*af*ph6 - 2*a0_a0*(5*af_p3 - 9*af_af*jMax*tf - 6*af*jMax*vd + 6*jMax_jMax*(-2*pd - tf*v0 + 3*tf*vf)) - 12*jMax_jMax*jMax*ph2 + a0*ph5)/(3*jMax_jMax*jMax*ph1);
polynom[4] := -(-a0_p6 - af_p6 + 6*a0_p5*(af - jMax*tf) - 48*af_p3*jMax_jMax*g1 + 72*jMax_jMax*jMax*(jMax*g1*g1 + vd_vd*vd + 2*af*g1*vd) - 3*a0_p4*ph3 - 36*af_af*jMax_jMax*vd_vd + 6*af_p4*jMax*vd + 4*a0_p3*(5*af_p3 - 9*af_af*jMax*tf - 6*af*jMax*vd + 6*jMax_jMax*(-2*pd - tf*v0 + 3*tf*vf)) - 3*a0_a0*ph5 + 6*a0*(af_p5 - af_p4*jMax*tf - 4*af_p3*jMax*(jMax*tf_tf + vd) + 12*jMax_jMax*(-af*ph6 + jMax*ph2)))/(18*jMax_jMax*jMax_jMax*ph1);

Roots.SolveQuartMonic(ADR(polynom[1]), 4, rootCount:=d_extremasCount, roots:=d_extremas);
t_max := (a0 - aMin)/jMax;
FOR i:=0 TO d_extremasCount
DO
  t := d_extremas[i];
  IF t > t_max
  THEN
    CONTINUE;
  END_IF

  // Single Newton step (regarding pd)
  h1 := ad_ad/2 + jMax*(af*t + (jMax*t - a0)*(t - tf) - vd);
  h2 := -ad + jMax*(tf - 2*t);
  IF h1 < 0
  THEN
    CONTINUE;
  END_IF
  
  h3 := SQRT(h1);
  orig := (af_p3 - a0_p3 + 3*af*jMax*t*(af + jMax*t) + 3*a0_a0*(af + jMax*t) - 3*a0*(af_af + 2*af*jMax*t + jMax_jMax*(t*t - tf_tf)) + 3*jMax_jMax*(-2*pd + jMax*t*(t - tf)*tf + 2*tf*v0))/(6*jMax_jMax) - h3*h3*h3/(jMax*ABS(jMax)) + ((-ad - jMax*t)*h1)/(jMax_jMax);
  deriv := (6*jMax*h2*h3/ABS(jMax) + 2*(-ad - jMax*tf)*h2 - 2*(3*ad_ad + af*jMax*(8*t - 2*tf) + 4*a0*jMax*(-2*t + tf) + 2*jMax*(jMax*t*(3*t - 2*tf) - vd)))/(4*jMax);
  t := t - orig / deriv;
  
  h1 := 2*ad_ad + 4*jMax*(ad*t + a0*tf + jMax*t*(t - tf) - vd);
  IF h1 < 0
  THEN
    CONTINUE;
	END_IF
  
  h1 := SQRT(h1)/ABS(jMax);
  
  // Solution 2 with aPlat
  Profile.t[0] := 0;
  Profile.t[1] := 0;
  Profile.t[2] := t;
  Profile.t[3] := tf - 2*t - ad/jMax - h1;
  Profile.t[4] := h1*0.5;
  Profile.t[5] := 0;
  Profile.t[6] := tf - (t + Profile.t[3] + Profile.t[4]);
  
  time_none := Profile.CheckWithTiming(ProfileJerkSigns.Uddu, ProfileLimits.None, tf, jMax, vMax, vMin, aMax, aMin);
  IF time_none
  THEN
    RETURN;
  END_IF
END_FOR

// Profiles with a3 != 0, Solution UDUD
// T 0124
ph0 := -2*pd - tf*v0 + 3*tf*vf;
ph1 := -ad + jMax*tf;
ph2 := jMax*tf_tf*g1 - vd*ph0;
ph3 := 5*af_af + 2*jMax*(2*jMax*tf_tf - vd - 4*af*tf);
ph4 := jMax_jMax*tf_p4 - 2*vd_vd + 8*jMax*tf*(-pd + tf*vf);
ph5 := (5*af_p4 - 8*af_p3*jMax*tf - 12*af_af*jMax*(jMax*tf_tf + vd) + 24*af*jMax_jMax*(-2*pd + jMax*tf_p3 + 2*tf*vf) - 6*jMax_jMax*ph4);
ph6 := -vd_vd + jMax*tf*(-2*pd + 3*tf*v0 - tf*vf);
ph7 := 3*jMax_jMax*ph1*ph1;

polynom[1] := (4*af*tf - 2*jMax*tf_tf - 4*vd)/ph1;
polynom[2] := (-2*(a0_p4 + af_p4) + 8*af_p3*jMax*tf + 6*af_af*jMax_jMax*tf_tf + 8*a0_p3*(af - jMax*tf) - 12*a0_a0*(af - jMax*tf)*(af - jMax*tf) - 12*af*jMax_jMax*(-pd + jMax*tf_p3 - 2*tf*v0 + 3*tf*vf) + 2*a0*(4*af_p3 - 12*af_af*jMax*tf + 9*af*jMax_jMax*tf_tf - 3*jMax_jMax*(2*pd + jMax*tf_p3 - 2*tf*vf)) + 3*jMax_jMax*(jMax_jMax*tf_p4 + 4*vd_vd - 4*jMax*tf*(pd + tf*v0 - 2*tf*vf)))/ph7;
polynom[3] := (-a0_p5 + af_p5 - af_p4*jMax*tf + 5*a0_p4*(af - jMax*tf) - 2*a0_p3*ph3 - 4*af_p3*jMax*(jMax*tf_tf + vd) + 12*af_af*jMax_jMax*g2 - 12*af*jMax_jMax*ph6 + 2*a0_a0*(5*af_p3 - 9*af_af*jMax*tf - 6*af*jMax*vd + 6*jMax_jMax*ph0) + 12*jMax_jMax*jMax*ph2 + a0*(-5*af_p4 + 8*af_p3*jMax*tf + 12*af_af*jMax*(jMax*tf_tf + vd) - 24*af*jMax_jMax*(-2*pd + jMax*tf_p3 + 2*tf*vf) + 6*jMax_jMax*ph4))/(jMax*ph7);
polynom[4] := -(a0_p6 + af_p6 - 6*a0_p5*(af - jMax*tf) + 48*af_p3*jMax_jMax*g1 - 72*jMax_jMax*jMax*(jMax*g1*g1 + vd_vd*vd + 2*af*g1*vd) + 3*a0_p4*ph3 - 6*af_p4*jMax*vd + 36*af_af*jMax_jMax*vd_vd - 4*a0_p3*(5*af_p3 - 9*af_af*jMax*tf - 6*af*jMax*vd + 6*jMax_jMax*ph0) + 3*a0_a0*ph5 - 6*a0*(af_p5 - af_p4*jMax*tf - 4*af_p3*jMax*(jMax*tf_tf + vd) + 12*jMax_jMax*(af_af*g2 - af*ph6 + jMax*ph2)))/(6*jMax_jMax*ph7);

Roots.SolveQuartMonic(ADR(polynom[1]), 4, rootCount:=d_extremasCount, roots:=d_extremas);
FOR i:=0 TO d_extremasCount
DO
  t := d_extremas[i];
  IF t > tf OR_ELSE t > (aMax - a0)/jMax
  THEN
    CONTINUE;
	END_IF

  h1 := ad_ad/(2*jMax_jMax) + (a0*(t + tf) - af*t + jMax*t*tf - vd)/jMax;
  IF h1 >= 0
  THEN
    h1 := SQRT(h1);
    
    Profile.t[0] := t;
    Profile.t[1] := tf - ad/jMax - 2*h1;
    Profile.t[2] := h1;
    Profile.t[3] := 0;
    Profile.t[4] := ad/jMax + h1 - t;
    Profile.t[5] := 0;
    Profile.t[6] := 0;
  
